% RSLogix 500 project HB_1_Filler.RSS, saved by version 12.00.00.00 %
PROJECT "PLC"    % processor: MicroLogix 1400 %

PROGRAM FILES
  LAD 2 "MAIN"  23 rungs
  LAD 9 "DPSTR REAR"  42 rungs
  LAD 11 "MAP DI"  37 rungs
  LAD 12 "MAP DO"  17 rungs
  LAD 14 "ALARMS"  17 rungs

DATA FILES
  O0 OUTPUT  7 elements
  I1 INPUT  9 elements
  S2 STATUS  66 elements
  B3 BINARY  14 elements
  T4 TIMER  22 elements
  C5 COUNTER  10 elements
  R6 CONTROL  5 elements
  N7 INTEGER  50 elements
  F8 FLOAT  40 elements
  B11 MAP DI  5 elements
  B12 MAP DO  10 elements
  B13 FORCE OUT  10 elements
  B23 TYPICAL  30 elements
  T24 TYPICAL  90 elements
  C25 TYPICAL  10 elements
  N27 TYPICAL  200 elements
  F28 TYPICAL  40 elements

LADDER 2 "MAIN"
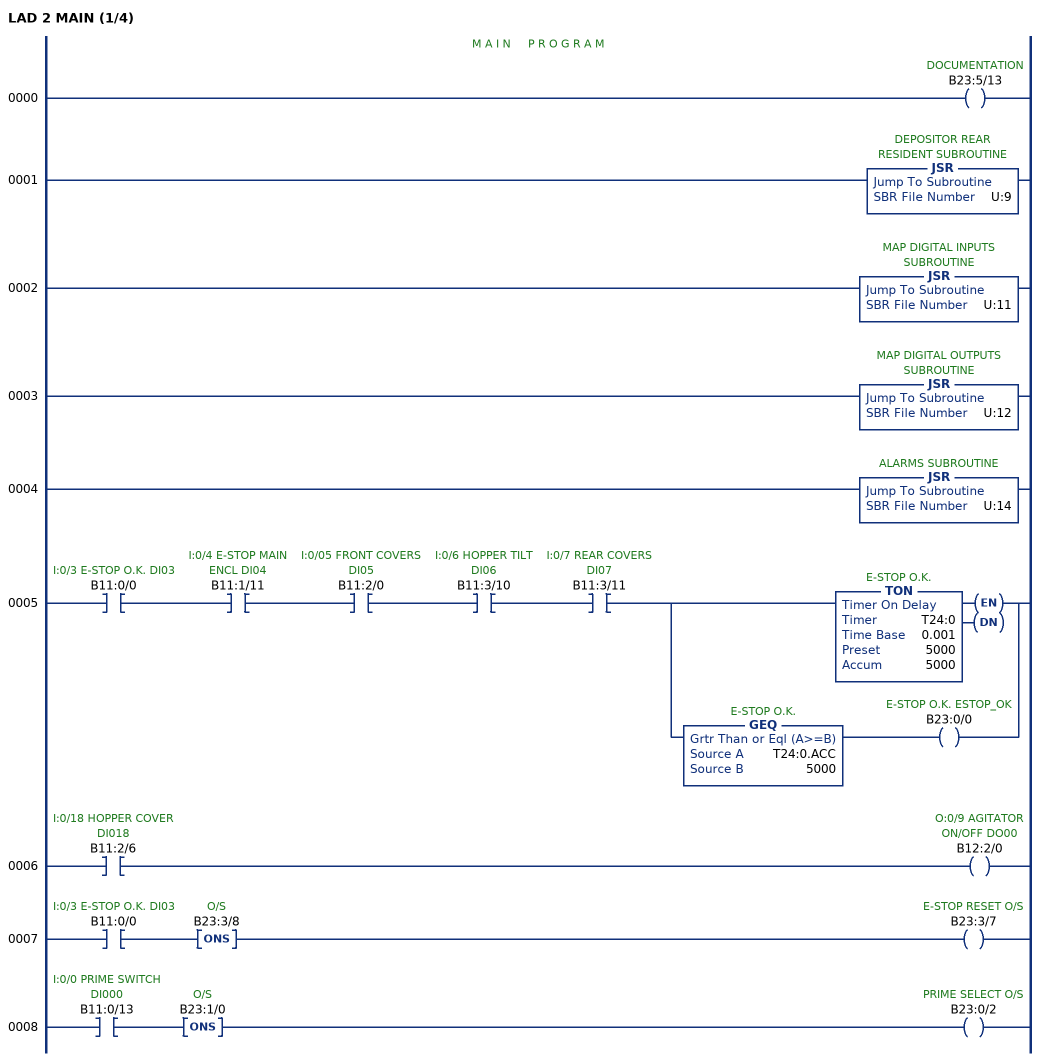
% Rung: 0 %
%  M A I N     P R O G R A M %
SOR OTE B23:5/13 EOR
%   B23:5/13  "DOCUMENTATION" %
% Rung: 1 %
SOR JSR U:9 EOR
%   U:9  "DEPOSITOR REAR RESIDENT SUBROUTINE" %
% Rung: 2 %
SOR JSR U:11 EOR
%   U:11  "MAP DIGITAL INPUTS SUBROUTINE" %
% Rung: 3 %
SOR JSR U:12 EOR
%   U:12  "MAP DIGITAL OUTPUTS SUBROUTINE" %
% Rung: 4 %
SOR JSR U:14 EOR
%   U:14  "ALARMS SUBROUTINE" %
% Rung: 5 %
SOR XIC B11:0/0 XIC B11:1/11 XIC B11:2/0 XIC B11:3/10 XIC B11:3/11 BST TON T24:0 0.001 5000 5000 NXB GEQ T24:0.ACC 5000 OTE B23:0/0 BND EOR
%   B11:0/0  DI03  "I:0/3 E-STOP O.K." %
%   B11:1/11  DI04  "I:0/4 E-STOP MAIN ENCL" %
%   B11:2/0  DI05  "I:0/05 FRONT COVERS" %
%   B11:3/10  DI06  "I:0/6 HOPPER TILT" %
%   B11:3/11  DI07  "I:0/7 REAR COVERS" %
%   T24:0  "E-STOP O.K." %
%   B23:0/0  ESTOP_OK  "E-STOP O.K." %
% Rung: 6 %
SOR XIC B11:2/6 OTE B12:2/0 EOR
%   B11:2/6  DI018  "I:0/18 HOPPER COVER" %
%   B12:2/0  DO00  "O:0/9 AGITATOR ON/OFF" %
% Rung: 7 %
SOR XIC B11:0/0 ONS B23:3/8 OTE B23:3/7 EOR
%   B11:0/0  DI03  "I:0/3 E-STOP O.K." %
%   B23:3/8  "O/S" %
%   B23:3/7  "E-STOP RESET O/S" %
% Rung: 8 %
SOR XIC B11:0/13 ONS B23:1/0 OTE B23:0/2 EOR
%   B11:0/13  DI000  "I:0/0 PRIME SWITCH" %
%   B23:1/0  "O/S" %
%   B23:0/2  "PRIME SELECT O/S" %

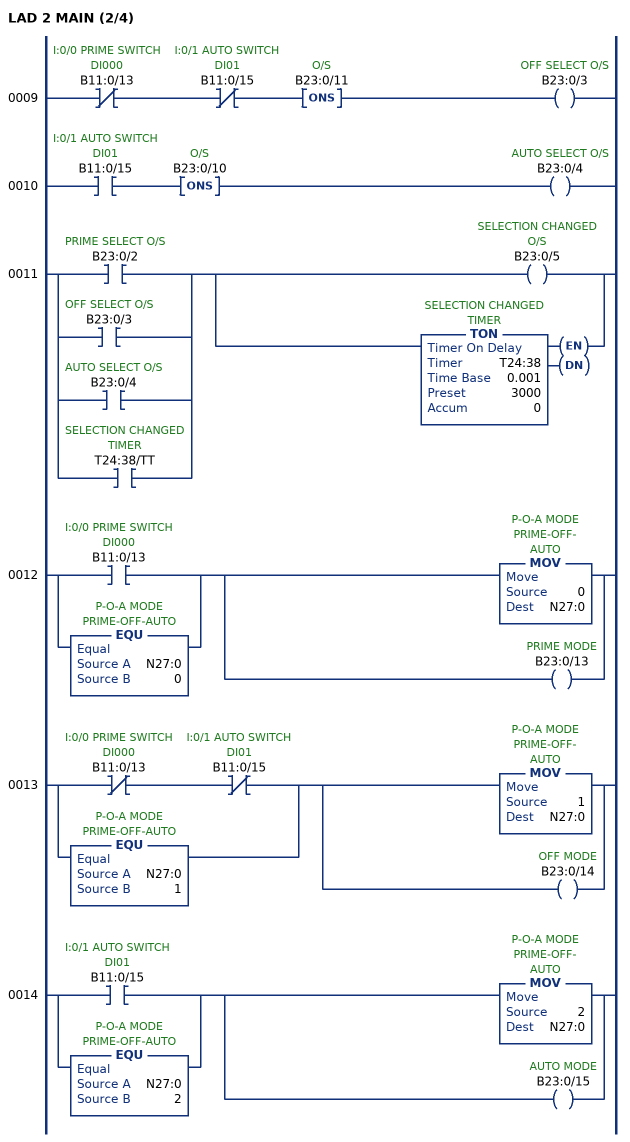
% Rung: 9 %
SOR XIO B11:0/13 XIO B11:0/15 ONS B23:0/11 OTE B23:0/3 EOR
%   B11:0/13  DI000  "I:0/0 PRIME SWITCH" %
%   B11:0/15  DI01  "I:0/1 AUTO SWITCH" %
%   B23:0/11  "O/S" %
%   B23:0/3  "OFF SELECT O/S" %
% Rung: 10 %
SOR XIC B11:0/15 ONS B23:0/10 OTE B23:0/4 EOR
%   B11:0/15  DI01  "I:0/1 AUTO SWITCH" %
%   B23:0/10  "O/S" %
%   B23:0/4  "AUTO SELECT O/S" %
% Rung: 11 %
SOR BST XIC B23:0/2 NXB XIC B23:0/3 NXB XIC B23:0/4 NXB XIC T24:38/TT BND BST OTE B23:0/5 NXB TON T24:38 0.001 3000 0 BND EOR
%   B23:0/2  "PRIME SELECT O/S" %
%   B23:0/3  "OFF SELECT O/S" %
%   B23:0/4  "AUTO SELECT O/S" %
%   T24:38  "SELECTION CHANGED TIMER" %
%   B23:0/5  "SELECTION CHANGED O/S" %
% Rung: 12 %
SOR BST XIC B11:0/13 NXB EQU N27:0 0 BND BST MOV 0 N27:0 NXB OTE B23:0/13 BND EOR
%   B11:0/13  DI000  "I:0/0 PRIME SWITCH" %
%   N27:0  "P-O-A MODE PRIME-OFF-AUTO" %
%   B23:0/13  "PRIME MODE" %
% Rung: 13 %
SOR BST XIO B11:0/13 XIO B11:0/15 NXB EQU N27:0 1 BND BST MOV 1 N27:0 NXB OTE B23:0/14 BND EOR
%   B11:0/13  DI000  "I:0/0 PRIME SWITCH" %
%   B11:0/15  DI01  "I:0/1 AUTO SWITCH" %
%   N27:0  "P-O-A MODE PRIME-OFF-AUTO" %
%   B23:0/14  "OFF MODE" %
% Rung: 14 %
SOR BST XIC B11:0/15 NXB EQU N27:0 2 BND BST MOV 2 N27:0 NXB OTE B23:0/15 BND EOR
%   B11:0/15  DI01  "I:0/1 AUTO SWITCH" %
%   N27:0  "P-O-A MODE PRIME-OFF-AUTO" %
%   B23:0/15  "AUTO MODE" %

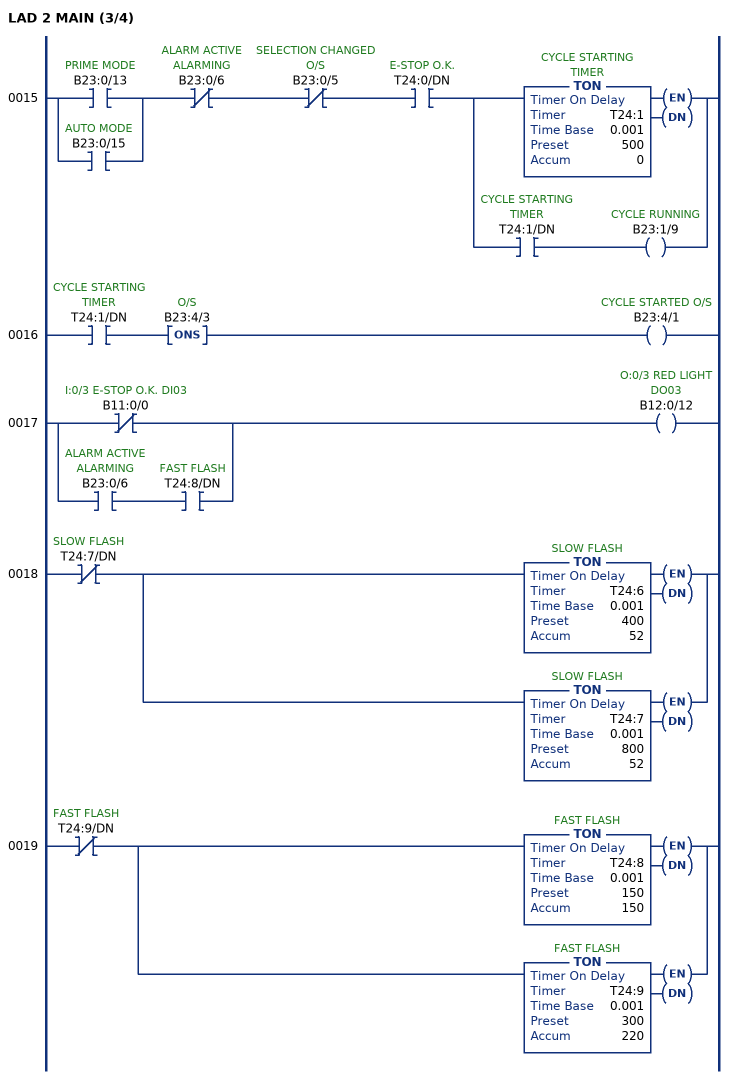
% Rung: 15 %
SOR BST XIC B23:0/13 NXB XIC B23:0/15 BND XIO B23:0/6 XIO B23:0/5 XIC T24:0/DN BST TON T24:1 0.001 500 0 NXB XIC T24:1/DN OTE B23:1/9 BND EOR
%   B23:0/13  "PRIME MODE" %
%   B23:0/15  "AUTO MODE" %
%   B23:0/6  ALARMING  "ALARM ACTIVE" %
%   B23:0/5  "SELECTION CHANGED O/S" %
%   T24:0  "E-STOP O.K." %
%   T24:1  "CYCLE STARTING TIMER" %
%   B23:1/9  "CYCLE RUNNING" %
% Rung: 16 %
SOR XIC T24:1/DN ONS B23:4/3 OTE B23:4/1 EOR
%   T24:1  "CYCLE STARTING TIMER" %
%   B23:4/3  "O/S" %
%   B23:4/1  "CYCLE STARTED O/S" %
% Rung: 17 %
SOR BST XIO B11:0/0 NXB XIC B23:0/6 XIC T24:8/DN BND OTE B12:0/12 EOR
%   B11:0/0  DI03  "I:0/3 E-STOP O.K." %
%   B23:0/6  ALARMING  "ALARM ACTIVE" %
%   T24:8  "FAST FLASH" %
%   B12:0/12  DO03  "O:0/3 RED LIGHT" %
% Rung: 18 %
SOR XIO T24:7/DN BST TON T24:6 0.001 400 52 NXB TON T24:7 0.001 800 52 BND EOR
%   T24:7  "SLOW FLASH" %
%   T24:6  "SLOW FLASH" %
% Rung: 19 %
SOR XIO T24:9/DN BST TON T24:8 0.001 150 150 NXB TON T24:9 0.001 300 220 BND EOR
%   T24:9  "FAST FLASH" %
%   T24:8  "FAST FLASH" %

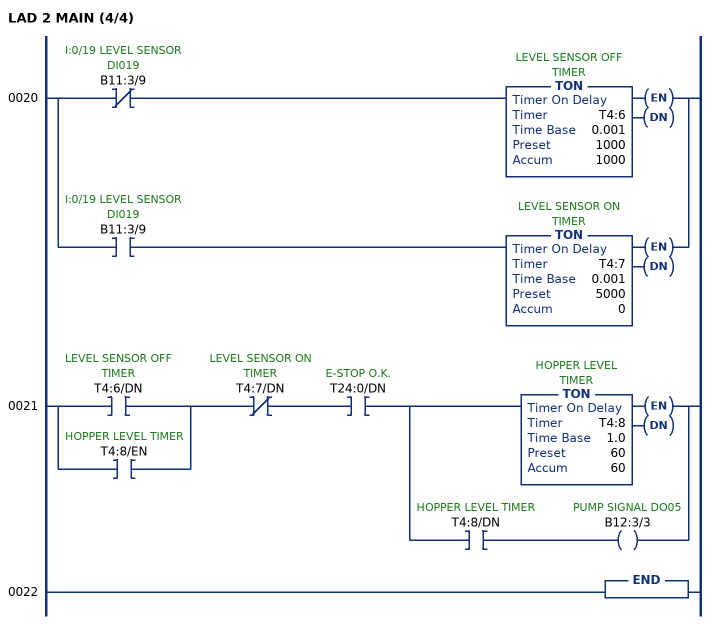
% Rung: 20 %
SOR BST XIO B11:3/9 TON T4:6 0.001 1000 1000 NXB XIC B11:3/9 TON T4:7 0.001 5000 0 BND EOR
%   B11:3/9  DI019  "I:0/19 LEVEL SENSOR" %
%   T4:6  "LEVEL SENSOR OFF TIMER" %
%   T4:7  "LEVEL SENSOR ON TIMER" %
% Rung: 21 %
SOR BST XIC T4:6/DN NXB XIC T4:8/EN BND XIO T4:7/DN XIC T24:0/DN BST TON T4:8 1.0 60 60 NXB XIC T4:8/DN OTE B12:3/3 BND EOR
%   T4:6  "LEVEL SENSOR OFF TIMER" %
%   T4:8  "HOPPER LEVEL TIMER" %
%   T4:7  "LEVEL SENSOR ON TIMER" %
%   T24:0  "E-STOP O.K." %
%   B12:3/3  DO05  "PUMP SIGNAL" %
% Rung: 22 %
SOR END EOR

LADDER 9 "DPSTR REAR"
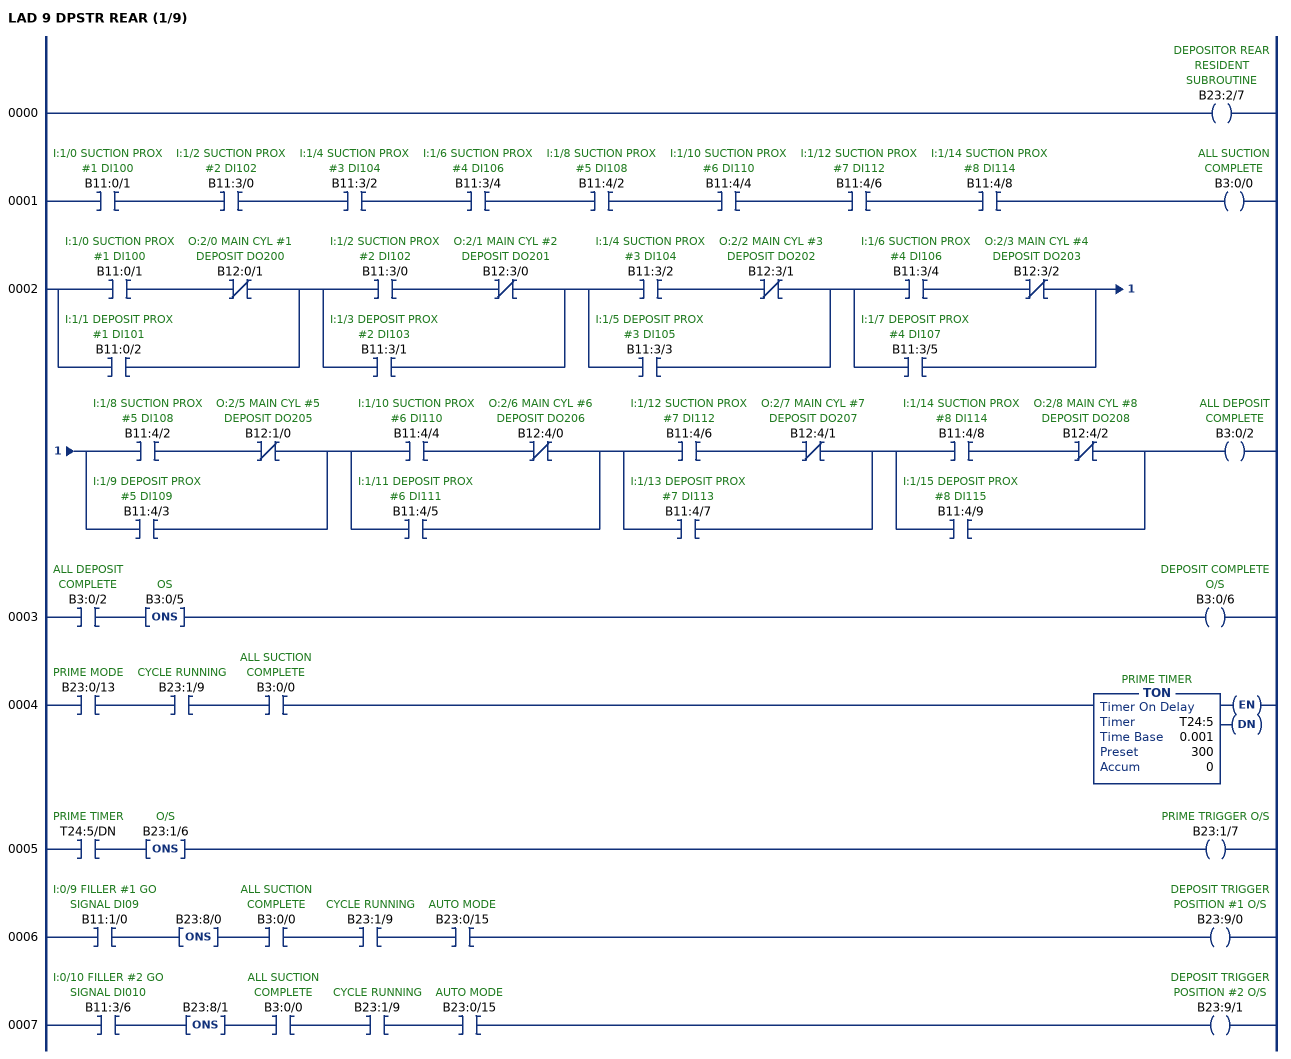
% Rung: 0 %
SOR OTE B23:2/7 EOR
%   B23:2/7  "DEPOSITOR REAR RESIDENT SUBROUTINE" %
% Rung: 1 %
SOR XIC B11:0/1 XIC B11:3/0 XIC B11:3/2 XIC B11:3/4 XIC B11:4/2 XIC B11:4/4 XIC B11:4/6 XIC B11:4/8 OTE B3:0/0 EOR
%   B11:0/1  DI100  "I:1/0 SUCTION PROX #1" %
%   B11:3/0  DI102  "I:1/2 SUCTION PROX #2" %
%   B11:3/2  DI104  "I:1/4 SUCTION PROX #3" %
%   B11:3/4  DI106  "I:1/6 SUCTION PROX #4" %
%   B11:4/2  DI108  "I:1/8 SUCTION PROX #5" %
%   B11:4/4  DI110  "I:1/10 SUCTION PROX #6" %
%   B11:4/6  DI112  "I:1/12 SUCTION PROX #7" %
%   B11:4/8  DI114  "I:1/14 SUCTION PROX #8" %
%   B3:0/0  "ALL SUCTION COMPLETE" %
% Rung: 2 %
SOR BST XIC B11:0/1 XIO B12:0/1 NXB XIC B11:0/2 BND BST XIC B11:3/0 XIO B12:3/0 NXB XIC B11:3/1 BND BST XIC B11:3/2 XIO B12:3/1 NXB XIC B11:3/3 BND BST XIC B11:3/4 XIO B12:3/2 NXB XIC B11:3/5 BND BST XIC B11:4/2 XIO B12:1/0 NXB XIC B11:4/3 BND BST XIC B11:4/4 XIO B12:4/0 NXB XIC B11:4/5 BND BST XIC B11:4/6 XIO B12:4/1 NXB XIC B11:4/7 BND BST XIC B11:4/8 XIO B12:4/2 NXB XIC B11:4/9 BND OTE B3:0/2 EOR
%   B11:0/1  DI100  "I:1/0 SUCTION PROX #1" %
%   B12:0/1  DO200  "O:2/0 MAIN CYL #1 DEPOSIT" %
%   B11:0/2  DI101  "I:1/1 DEPOSIT PROX #1" %
%   B11:3/0  DI102  "I:1/2 SUCTION PROX #2" %
%   B12:3/0  DO201  "O:2/1 MAIN CYL #2 DEPOSIT" %
%   B11:3/1  DI103  "I:1/3 DEPOSIT PROX #2" %
%   B11:3/2  DI104  "I:1/4 SUCTION PROX #3" %
%   B12:3/1  DO202  "O:2/2 MAIN CYL #3 DEPOSIT" %
%   B11:3/3  DI105  "I:1/5 DEPOSIT PROX #3" %
%   B11:3/4  DI106  "I:1/6 SUCTION PROX #4" %
%   B12:3/2  DO203  "O:2/3 MAIN CYL #4 DEPOSIT" %
%   B11:3/5  DI107  "I:1/7 DEPOSIT PROX #4" %
%   B11:4/2  DI108  "I:1/8 SUCTION PROX #5" %
%   B12:1/0  DO205  "O:2/5 MAIN CYL #5 DEPOSIT" %
%   B11:4/3  DI109  "I:1/9 DEPOSIT PROX #5" %
%   B11:4/4  DI110  "I:1/10 SUCTION PROX #6" %
%   B12:4/0  DO206  "O:2/6 MAIN CYL #6 DEPOSIT" %
%   B11:4/5  DI111  "I:1/11 DEPOSIT PROX #6" %
%   B11:4/6  DI112  "I:1/12 SUCTION PROX #7" %
%   B12:4/1  DO207  "O:2/7 MAIN CYL #7 DEPOSIT" %
%   B11:4/7  DI113  "I:1/13 DEPOSIT PROX #7" %
%   B11:4/8  DI114  "I:1/14 SUCTION PROX #8" %
%   B12:4/2  DO208  "O:2/8 MAIN CYL #8 DEPOSIT" %
%   B11:4/9  DI115  "I:1/15 DEPOSIT PROX #8" %
%   B3:0/2  "ALL DEPOSIT COMPLETE" %
% Rung: 3 %
SOR XIC B3:0/2 ONS B3:0/5 OTE B3:0/6 EOR
%   B3:0/2  "ALL DEPOSIT COMPLETE" %
%   B3:0/5  "OS" %
%   B3:0/6  "DEPOSIT COMPLETE O/S" %
% Rung: 4 %
SOR XIC B23:0/13 XIC B23:1/9 XIC B3:0/0 TON T24:5 0.001 300 0 EOR
%   B23:0/13  "PRIME MODE" %
%   B23:1/9  "CYCLE RUNNING" %
%   B3:0/0  "ALL SUCTION COMPLETE" %
%   T24:5  "PRIME TIMER" %
% Rung: 5 %
SOR XIC T24:5/DN ONS B23:1/6 OTE B23:1/7 EOR
%   T24:5  "PRIME TIMER" %
%   B23:1/6  "O/S" %
%   B23:1/7  "PRIME TRIGGER O/S" %
% Rung: 6 %
SOR XIC B11:1/0 ONS B23:8/0 XIC B3:0/0 XIC B23:1/9 XIC B23:0/15 OTE B23:9/0 EOR
%   B11:1/0  DI09  "I:0/9 FILLER #1 GO SIGNAL" %
%   B3:0/0  "ALL SUCTION COMPLETE" %
%   B23:1/9  "CYCLE RUNNING" %
%   B23:0/15  "AUTO MODE" %
%   B23:9/0  "DEPOSIT TRIGGER POSITION #1 O/S" %
% Rung: 7 %
SOR XIC B11:3/6 ONS B23:8/1 XIC B3:0/0 XIC B23:1/9 XIC B23:0/15 OTE B23:9/1 EOR
%   B11:3/6  DI010  "I:0/10 FILLER #2 GO SIGNAL" %
%   B3:0/0  "ALL SUCTION COMPLETE" %
%   B23:1/9  "CYCLE RUNNING" %
%   B23:0/15  "AUTO MODE" %
%   B23:9/1  "DEPOSIT TRIGGER POSITION #2 O/S" %

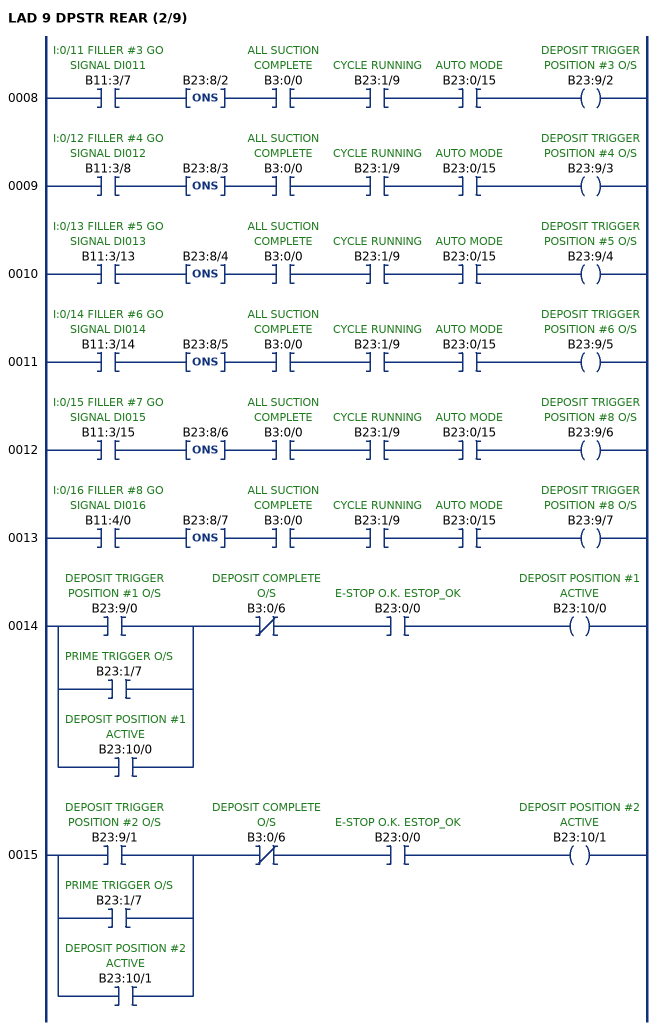
% Rung: 8 %
SOR XIC B11:3/7 ONS B23:8/2 XIC B3:0/0 XIC B23:1/9 XIC B23:0/15 OTE B23:9/2 EOR
%   B11:3/7  DI011  "I:0/11 FILLER #3 GO SIGNAL" %
%   B3:0/0  "ALL SUCTION COMPLETE" %
%   B23:1/9  "CYCLE RUNNING" %
%   B23:0/15  "AUTO MODE" %
%   B23:9/2  "DEPOSIT TRIGGER POSITION #3 O/S" %
% Rung: 9 %
SOR XIC B11:3/8 ONS B23:8/3 XIC B3:0/0 XIC B23:1/9 XIC B23:0/15 OTE B23:9/3 EOR
%   B11:3/8  DI012  "I:0/12 FILLER #4 GO SIGNAL" %
%   B3:0/0  "ALL SUCTION COMPLETE" %
%   B23:1/9  "CYCLE RUNNING" %
%   B23:0/15  "AUTO MODE" %
%   B23:9/3  "DEPOSIT TRIGGER POSITION #4 O/S" %
% Rung: 10 %
SOR XIC B11:3/13 ONS B23:8/4 XIC B3:0/0 XIC B23:1/9 XIC B23:0/15 OTE B23:9/4 EOR
%   B11:3/13  DI013  "I:0/13 FILLER #5 GO SIGNAL" %
%   B3:0/0  "ALL SUCTION COMPLETE" %
%   B23:1/9  "CYCLE RUNNING" %
%   B23:0/15  "AUTO MODE" %
%   B23:9/4  "DEPOSIT TRIGGER POSITION #5 O/S" %
% Rung: 11 %
SOR XIC B11:3/14 ONS B23:8/5 XIC B3:0/0 XIC B23:1/9 XIC B23:0/15 OTE B23:9/5 EOR
%   B11:3/14  DI014  "I:0/14 FILLER #6 GO SIGNAL" %
%   B3:0/0  "ALL SUCTION COMPLETE" %
%   B23:1/9  "CYCLE RUNNING" %
%   B23:0/15  "AUTO MODE" %
%   B23:9/5  "DEPOSIT TRIGGER POSITION #6 O/S" %
% Rung: 12 %
SOR XIC B11:3/15 ONS B23:8/6 XIC B3:0/0 XIC B23:1/9 XIC B23:0/15 OTE B23:9/6 EOR
%   B11:3/15  DI015  "I:0/15 FILLER #7 GO SIGNAL" %
%   B3:0/0  "ALL SUCTION COMPLETE" %
%   B23:1/9  "CYCLE RUNNING" %
%   B23:0/15  "AUTO MODE" %
%   B23:9/6  "DEPOSIT TRIGGER POSITION #8 O/S" %
% Rung: 13 %
SOR XIC B11:4/0 ONS B23:8/7 XIC B3:0/0 XIC B23:1/9 XIC B23:0/15 OTE B23:9/7 EOR
%   B11:4/0  DI016  "I:0/16 FILLER #8 GO SIGNAL" %
%   B3:0/0  "ALL SUCTION COMPLETE" %
%   B23:1/9  "CYCLE RUNNING" %
%   B23:0/15  "AUTO MODE" %
%   B23:9/7  "DEPOSIT TRIGGER POSITION #8 O/S" %
% Rung: 14 %
SOR BST XIC B23:9/0 NXB XIC B23:1/7 NXB XIC B23:10/0 BND XIO B3:0/6 XIC B23:0/0 OTE B23:10/0 EOR
%   B23:9/0  "DEPOSIT TRIGGER POSITION #1 O/S" %
%   B23:1/7  "PRIME TRIGGER O/S" %
%   B23:10/0  "DEPOSIT POSITION #1 ACTIVE" %
%   B3:0/6  "DEPOSIT COMPLETE O/S" %
%   B23:0/0  ESTOP_OK  "E-STOP O.K." %
% Rung: 15 %
SOR BST XIC B23:9/1 NXB XIC B23:1/7 NXB XIC B23:10/1 BND XIO B3:0/6 XIC B23:0/0 OTE B23:10/1 EOR
%   B23:9/1  "DEPOSIT TRIGGER POSITION #2 O/S" %
%   B23:1/7  "PRIME TRIGGER O/S" %
%   B23:10/1  "DEPOSIT POSITION #2 ACTIVE" %
%   B3:0/6  "DEPOSIT COMPLETE O/S" %
%   B23:0/0  ESTOP_OK  "E-STOP O.K." %

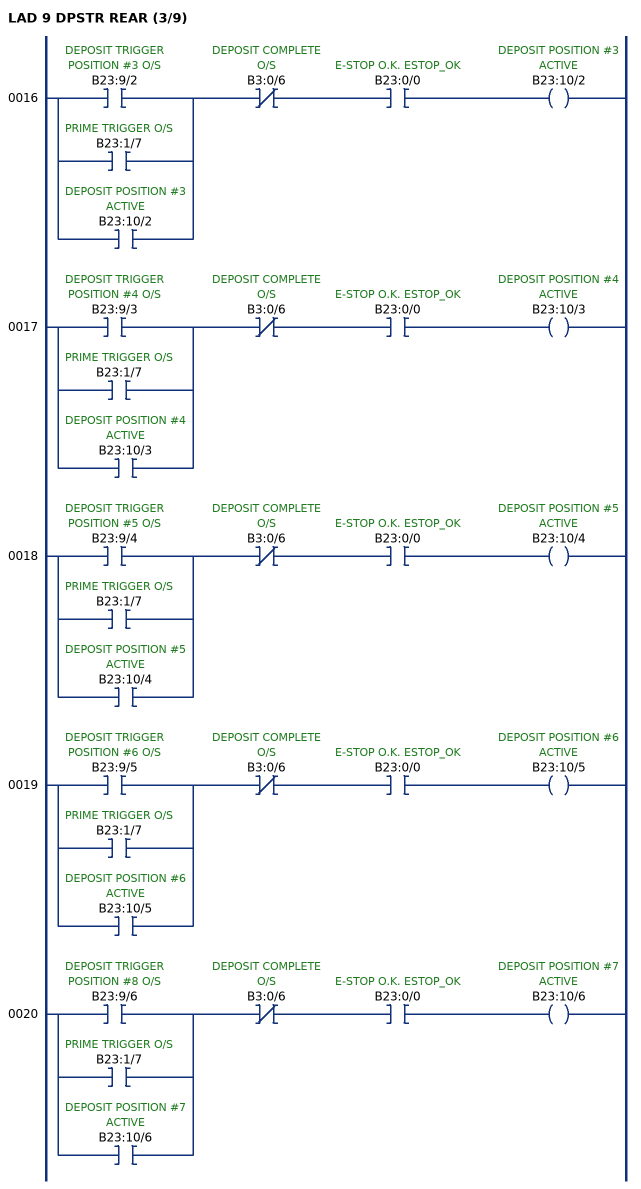
% Rung: 16 %
SOR BST XIC B23:9/2 NXB XIC B23:1/7 NXB XIC B23:10/2 BND XIO B3:0/6 XIC B23:0/0 OTE B23:10/2 EOR
%   B23:9/2  "DEPOSIT TRIGGER POSITION #3 O/S" %
%   B23:1/7  "PRIME TRIGGER O/S" %
%   B23:10/2  "DEPOSIT POSITION #3 ACTIVE" %
%   B3:0/6  "DEPOSIT COMPLETE O/S" %
%   B23:0/0  ESTOP_OK  "E-STOP O.K." %
% Rung: 17 %
SOR BST XIC B23:9/3 NXB XIC B23:1/7 NXB XIC B23:10/3 BND XIO B3:0/6 XIC B23:0/0 OTE B23:10/3 EOR
%   B23:9/3  "DEPOSIT TRIGGER POSITION #4 O/S" %
%   B23:1/7  "PRIME TRIGGER O/S" %
%   B23:10/3  "DEPOSIT POSITION #4 ACTIVE" %
%   B3:0/6  "DEPOSIT COMPLETE O/S" %
%   B23:0/0  ESTOP_OK  "E-STOP O.K." %
% Rung: 18 %
SOR BST XIC B23:9/4 NXB XIC B23:1/7 NXB XIC B23:10/4 BND XIO B3:0/6 XIC B23:0/0 OTE B23:10/4 EOR
%   B23:9/4  "DEPOSIT TRIGGER POSITION #5 O/S" %
%   B23:1/7  "PRIME TRIGGER O/S" %
%   B23:10/4  "DEPOSIT POSITION #5 ACTIVE" %
%   B3:0/6  "DEPOSIT COMPLETE O/S" %
%   B23:0/0  ESTOP_OK  "E-STOP O.K." %
% Rung: 19 %
SOR BST XIC B23:9/5 NXB XIC B23:1/7 NXB XIC B23:10/5 BND XIO B3:0/6 XIC B23:0/0 OTE B23:10/5 EOR
%   B23:9/5  "DEPOSIT TRIGGER POSITION #6 O/S" %
%   B23:1/7  "PRIME TRIGGER O/S" %
%   B23:10/5  "DEPOSIT POSITION #6 ACTIVE" %
%   B3:0/6  "DEPOSIT COMPLETE O/S" %
%   B23:0/0  ESTOP_OK  "E-STOP O.K." %
% Rung: 20 %
SOR BST XIC B23:9/6 NXB XIC B23:1/7 NXB XIC B23:10/6 BND XIO B3:0/6 XIC B23:0/0 OTE B23:10/6 EOR
%   B23:9/6  "DEPOSIT TRIGGER POSITION #8 O/S" %
%   B23:1/7  "PRIME TRIGGER O/S" %
%   B23:10/6  "DEPOSIT POSITION #7 ACTIVE" %
%   B3:0/6  "DEPOSIT COMPLETE O/S" %
%   B23:0/0  ESTOP_OK  "E-STOP O.K." %

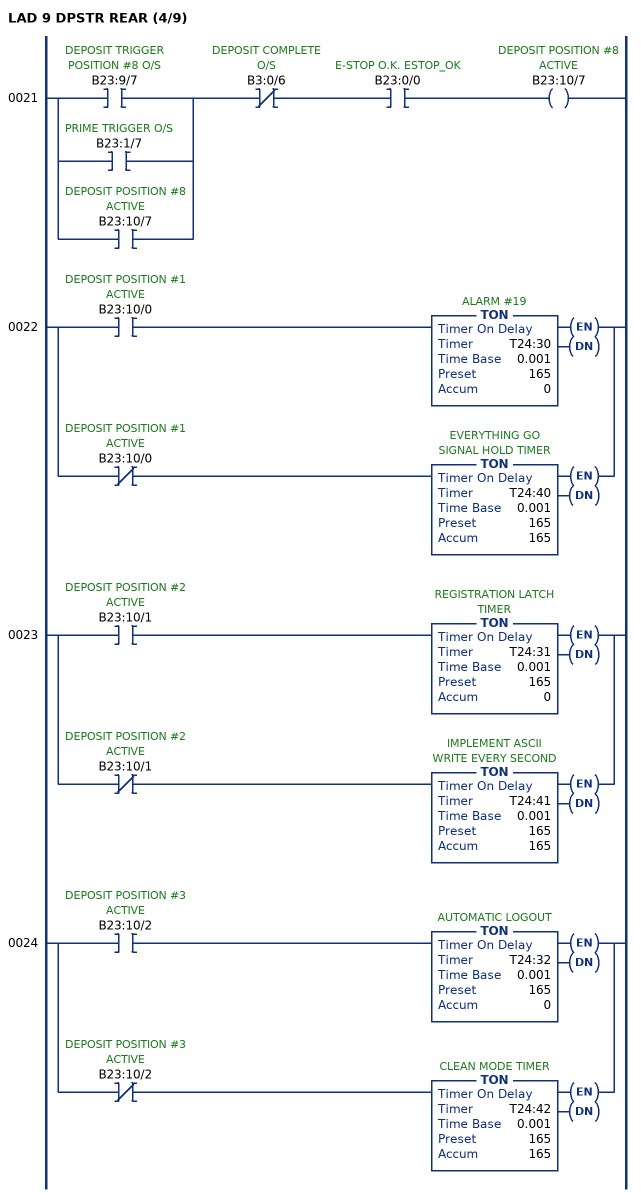
% Rung: 21 %
SOR BST XIC B23:9/7 NXB XIC B23:1/7 NXB XIC B23:10/7 BND XIO B3:0/6 XIC B23:0/0 OTE B23:10/7 EOR
%   B23:9/7  "DEPOSIT TRIGGER POSITION #8 O/S" %
%   B23:1/7  "PRIME TRIGGER O/S" %
%   B23:10/7  "DEPOSIT POSITION #8 ACTIVE" %
%   B3:0/6  "DEPOSIT COMPLETE O/S" %
%   B23:0/0  ESTOP_OK  "E-STOP O.K." %
% Rung: 22 %
SOR BST XIC B23:10/0 TON T24:30 0.001 165 0 NXB XIO B23:10/0 TON T24:40 0.001 165 165 BND EOR
%   B23:10/0  "DEPOSIT POSITION #1 ACTIVE" %
%   T24:30  "ALARM #19" %
%   T24:40  "EVERYTHING GO SIGNAL HOLD TIMER" %
% Rung: 23 %
SOR BST XIC B23:10/1 TON T24:31 0.001 165 0 NXB XIO B23:10/1 TON T24:41 0.001 165 165 BND EOR
%   B23:10/1  "DEPOSIT POSITION #2 ACTIVE" %
%   T24:31  "REGISTRATION LATCH TIMER" %
%   T24:41  "IMPLEMENT ASCII WRITE EVERY SECOND" %
% Rung: 24 %
SOR BST XIC B23:10/2 TON T24:32 0.001 165 0 NXB XIO B23:10/2 TON T24:42 0.001 165 165 BND EOR
%   B23:10/2  "DEPOSIT POSITION #3 ACTIVE" %
%   T24:32  "AUTOMATIC LOGOUT" %
%   T24:42  "CLEAN MODE TIMER" %

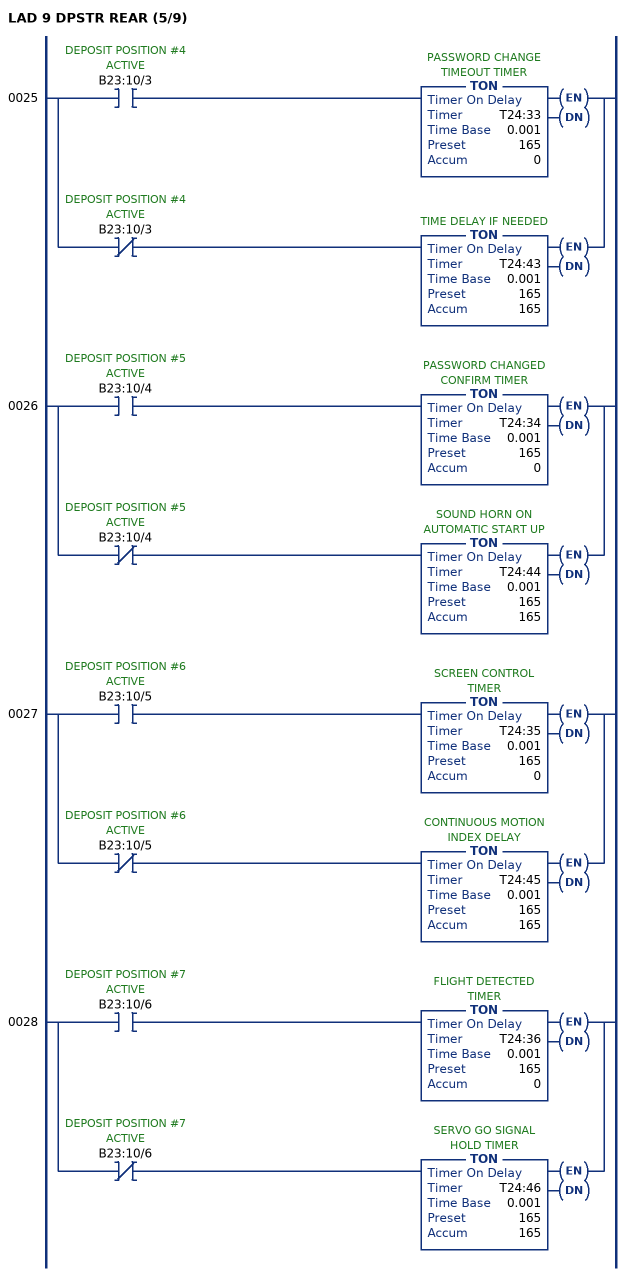
% Rung: 25 %
SOR BST XIC B23:10/3 TON T24:33 0.001 165 0 NXB XIO B23:10/3 TON T24:43 0.001 165 165 BND EOR
%   B23:10/3  "DEPOSIT POSITION #4 ACTIVE" %
%   T24:33  "PASSWORD CHANGE TIMEOUT TIMER" %
%   T24:43  "TIME DELAY IF NEEDED" %
% Rung: 26 %
SOR BST XIC B23:10/4 TON T24:34 0.001 165 0 NXB XIO B23:10/4 TON T24:44 0.001 165 165 BND EOR
%   B23:10/4  "DEPOSIT POSITION #5 ACTIVE" %
%   T24:34  "PASSWORD CHANGED CONFIRM TIMER" %
%   T24:44  "SOUND HORN ON AUTOMATIC START UP" %
% Rung: 27 %
SOR BST XIC B23:10/5 TON T24:35 0.001 165 0 NXB XIO B23:10/5 TON T24:45 0.001 165 165 BND EOR
%   B23:10/5  "DEPOSIT POSITION #6 ACTIVE" %
%   T24:35  "SCREEN CONTROL TIMER" %
%   T24:45  "CONTINUOUS MOTION INDEX DELAY" %
% Rung: 28 %
SOR BST XIC B23:10/6 TON T24:36 0.001 165 0 NXB XIO B23:10/6 TON T24:46 0.001 165 165 BND EOR
%   B23:10/6  "DEPOSIT POSITION #7 ACTIVE" %
%   T24:36  "FLIGHT DETECTED TIMER" %
%   T24:46  "SERVO GO SIGNAL HOLD TIMER" %

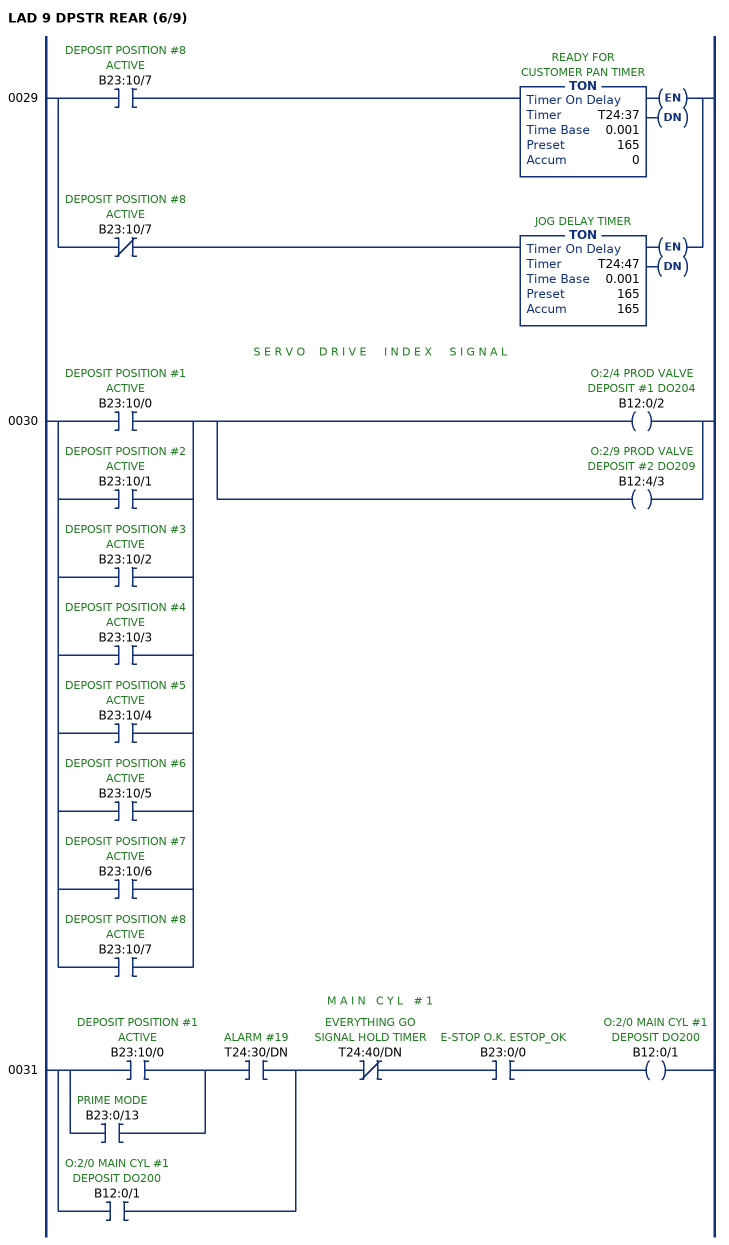
% Rung: 29 %
SOR BST XIC B23:10/7 TON T24:37 0.001 165 0 NXB XIO B23:10/7 TON T24:47 0.001 165 165 BND EOR
%   B23:10/7  "DEPOSIT POSITION #8 ACTIVE" %
%   T24:37  "READY FOR CUSTOMER PAN TIMER" %
%   T24:47  "JOG DELAY TIMER" %
% Rung: 30 %
%     S E R V O    D R I V E     I N D E X     S I G N A L %
SOR BST XIC B23:10/0 NXB XIC B23:10/1 NXB XIC B23:10/2 NXB XIC B23:10/3 NXB XIC B23:10/4 NXB XIC B23:10/5 NXB XIC B23:10/6 NXB XIC B23:10/7 BND BST OTE B12:0/2 NXB OTE B12:4/3 BND EOR
%   B23:10/0  "DEPOSIT POSITION #1 ACTIVE" %
%   B23:10/1  "DEPOSIT POSITION #2 ACTIVE" %
%   B23:10/2  "DEPOSIT POSITION #3 ACTIVE" %
%   B23:10/3  "DEPOSIT POSITION #4 ACTIVE" %
%   B23:10/4  "DEPOSIT POSITION #5 ACTIVE" %
%   B23:10/5  "DEPOSIT POSITION #6 ACTIVE" %
%   B23:10/6  "DEPOSIT POSITION #7 ACTIVE" %
%   B23:10/7  "DEPOSIT POSITION #8 ACTIVE" %
%   B12:0/2  DO204  "O:2/4 PROD VALVE DEPOSIT #1" %
%   B12:4/3  DO209  "O:2/9 PROD VALVE DEPOSIT #2" %
% Rung: 31 %
%     M A I N   C Y L   # 1 %
SOR BST BST XIC B23:10/0 NXB XIC B23:0/13 BND XIC T24:30/DN NXB XIC B12:0/1 BND XIO T24:40/DN XIC B23:0/0 OTE B12:0/1 EOR
%   B23:10/0  "DEPOSIT POSITION #1 ACTIVE" %
%   B23:0/13  "PRIME MODE" %
%   T24:30  "ALARM #19" %
%   B12:0/1  DO200  "O:2/0 MAIN CYL #1 DEPOSIT" %
%   T24:40  "EVERYTHING GO SIGNAL HOLD TIMER" %
%   B23:0/0  ESTOP_OK  "E-STOP O.K." %

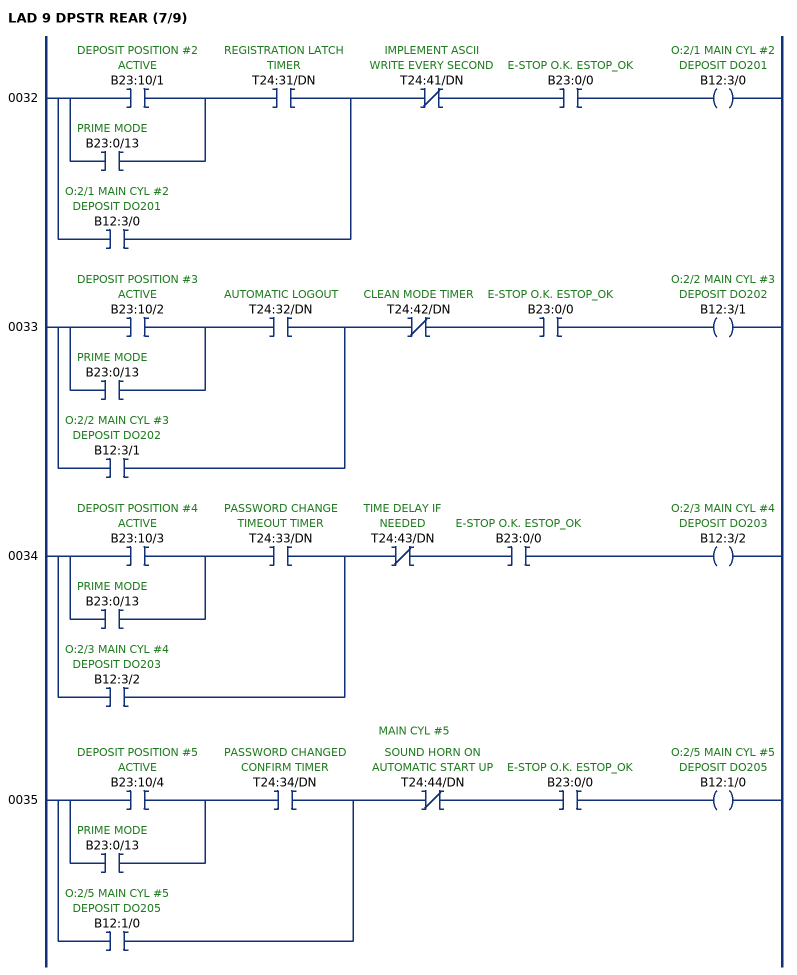
% Rung: 32 %
SOR BST BST XIC B23:10/1 NXB XIC B23:0/13 BND XIC T24:31/DN NXB XIC B12:3/0 BND XIO T24:41/DN XIC B23:0/0 OTE B12:3/0 EOR
%   B23:10/1  "DEPOSIT POSITION #2 ACTIVE" %
%   B23:0/13  "PRIME MODE" %
%   T24:31  "REGISTRATION LATCH TIMER" %
%   B12:3/0  DO201  "O:2/1 MAIN CYL #2 DEPOSIT" %
%   T24:41  "IMPLEMENT ASCII WRITE EVERY SECOND" %
%   B23:0/0  ESTOP_OK  "E-STOP O.K." %
% Rung: 33 %
SOR BST BST XIC B23:10/2 NXB XIC B23:0/13 BND XIC T24:32/DN NXB XIC B12:3/1 BND XIO T24:42/DN XIC B23:0/0 OTE B12:3/1 EOR
%   B23:10/2  "DEPOSIT POSITION #3 ACTIVE" %
%   B23:0/13  "PRIME MODE" %
%   T24:32  "AUTOMATIC LOGOUT" %
%   B12:3/1  DO202  "O:2/2 MAIN CYL #3 DEPOSIT" %
%   T24:42  "CLEAN MODE TIMER" %
%   B23:0/0  ESTOP_OK  "E-STOP O.K." %
% Rung: 34 %
SOR BST BST XIC B23:10/3 NXB XIC B23:0/13 BND XIC T24:33/DN NXB XIC B12:3/2 BND XIO T24:43/DN XIC B23:0/0 OTE B12:3/2 EOR
%   B23:10/3  "DEPOSIT POSITION #4 ACTIVE" %
%   B23:0/13  "PRIME MODE" %
%   T24:33  "PASSWORD CHANGE TIMEOUT TIMER" %
%   B12:3/2  DO203  "O:2/3 MAIN CYL #4 DEPOSIT" %
%   T24:43  "TIME DELAY IF NEEDED" %
%   B23:0/0  ESTOP_OK  "E-STOP O.K." %
% Rung: 35 %
% MAIN CYL #5 %
SOR BST BST XIC B23:10/4 NXB XIC B23:0/13 BND XIC T24:34/DN NXB XIC B12:1/0 BND XIO T24:44/DN XIC B23:0/0 OTE B12:1/0 EOR
%   B23:10/4  "DEPOSIT POSITION #5 ACTIVE" %
%   B23:0/13  "PRIME MODE" %
%   T24:34  "PASSWORD CHANGED CONFIRM TIMER" %
%   B12:1/0  DO205  "O:2/5 MAIN CYL #5 DEPOSIT" %
%   T24:44  "SOUND HORN ON AUTOMATIC START UP" %
%   B23:0/0  ESTOP_OK  "E-STOP O.K." %

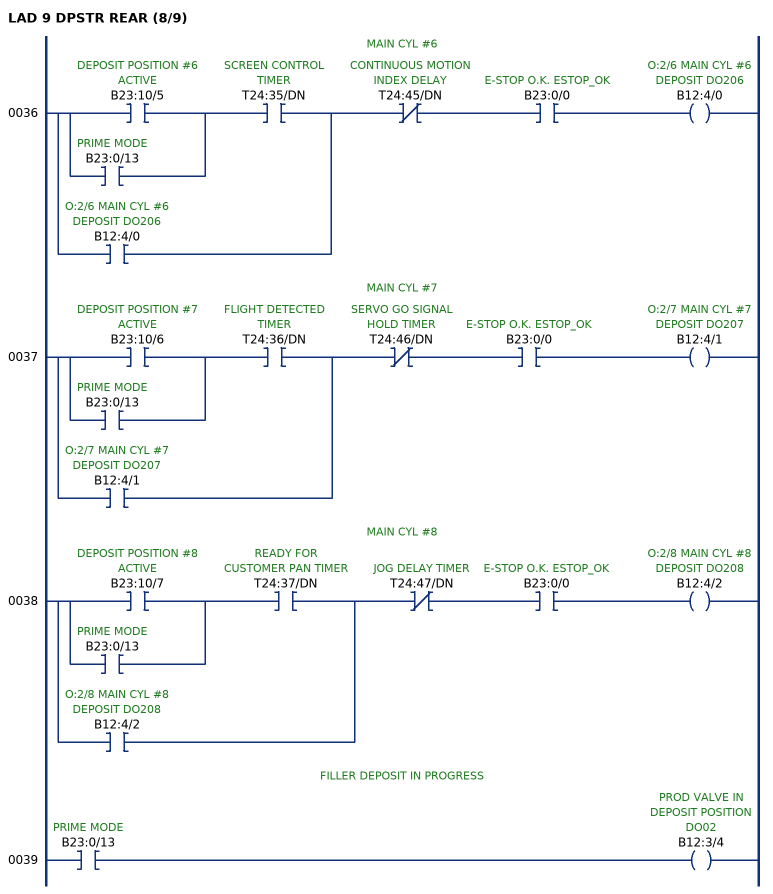
% Rung: 36 %
% MAIN CYL #6 %
SOR BST BST XIC B23:10/5 NXB XIC B23:0/13 BND XIC T24:35/DN NXB XIC B12:4/0 BND XIO T24:45/DN XIC B23:0/0 OTE B12:4/0 EOR
%   B23:10/5  "DEPOSIT POSITION #6 ACTIVE" %
%   B23:0/13  "PRIME MODE" %
%   T24:35  "SCREEN CONTROL TIMER" %
%   B12:4/0  DO206  "O:2/6 MAIN CYL #6 DEPOSIT" %
%   T24:45  "CONTINUOUS MOTION INDEX DELAY" %
%   B23:0/0  ESTOP_OK  "E-STOP O.K." %
% Rung: 37 %
% MAIN CYL #7 %
SOR BST BST XIC B23:10/6 NXB XIC B23:0/13 BND XIC T24:36/DN NXB XIC B12:4/1 BND XIO T24:46/DN XIC B23:0/0 OTE B12:4/1 EOR
%   B23:10/6  "DEPOSIT POSITION #7 ACTIVE" %
%   B23:0/13  "PRIME MODE" %
%   T24:36  "FLIGHT DETECTED TIMER" %
%   B12:4/1  DO207  "O:2/7 MAIN CYL #7 DEPOSIT" %
%   T24:46  "SERVO GO SIGNAL HOLD TIMER" %
%   B23:0/0  ESTOP_OK  "E-STOP O.K." %
% Rung: 38 %
% MAIN CYL #8 %
SOR BST BST XIC B23:10/7 NXB XIC B23:0/13 BND XIC T24:37/DN NXB XIC B12:4/2 BND XIO T24:47/DN XIC B23:0/0 OTE B12:4/2 EOR
%   B23:10/7  "DEPOSIT POSITION #8 ACTIVE" %
%   B23:0/13  "PRIME MODE" %
%   T24:37  "READY FOR CUSTOMER PAN TIMER" %
%   B12:4/2  DO208  "O:2/8 MAIN CYL #8 DEPOSIT" %
%   T24:47  "JOG DELAY TIMER" %
%   B23:0/0  ESTOP_OK  "E-STOP O.K." %
% Rung: 39 %
% FILLER DEPOSIT IN PROGRESS %
SOR XIC B23:0/13 OTE B12:3/4 EOR
%   B23:0/13  "PRIME MODE" %
%   B12:3/4  DO02  "PROD VALVE IN DEPOSIT POSITION" %

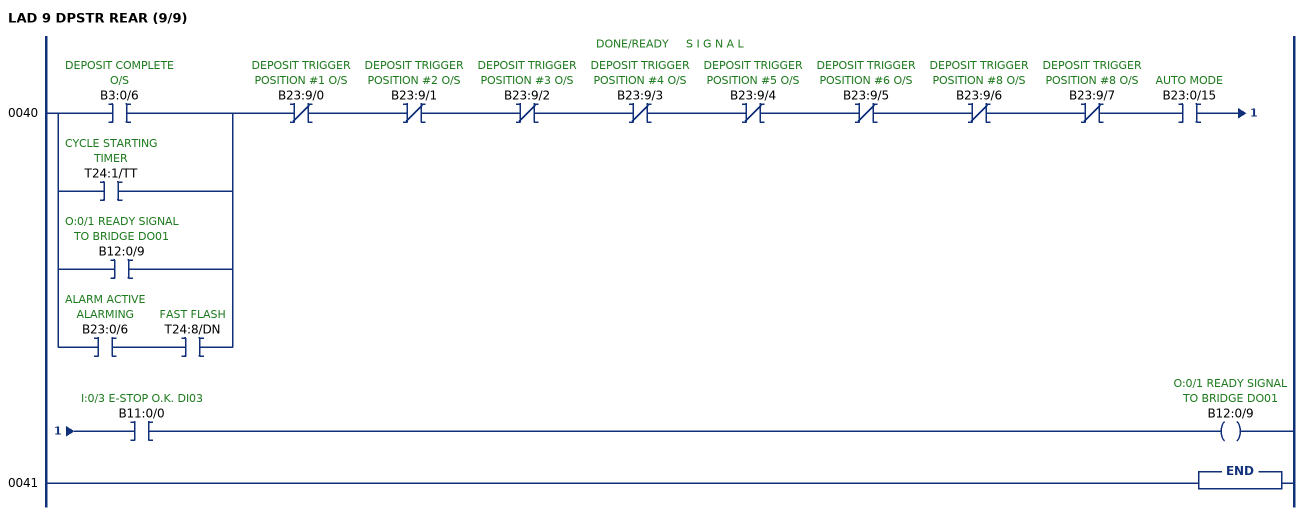
% Rung: 40 %
%         DONE/READY     S I G N A L %
SOR BST XIC B3:0/6 NXB XIC T24:1/TT NXB XIC B12:0/9 NXB XIC B23:0/6 XIC T24:8/DN BND XIO B23:9/0 XIO B23:9/1 XIO B23:9/2 XIO B23:9/3 XIO B23:9/4 XIO B23:9/5 XIO B23:9/6 XIO B23:9/7 XIC B23:0/15 XIC B11:0/0 OTE B12:0/9 EOR
%   B3:0/6  "DEPOSIT COMPLETE O/S" %
%   T24:1  "CYCLE STARTING TIMER" %
%   B12:0/9  DO01  "O:0/1 READY SIGNAL TO BRIDGE" %
%   B23:0/6  ALARMING  "ALARM ACTIVE" %
%   T24:8  "FAST FLASH" %
%   B23:9/0  "DEPOSIT TRIGGER POSITION #1 O/S" %
%   B23:9/1  "DEPOSIT TRIGGER POSITION #2 O/S" %
%   B23:9/2  "DEPOSIT TRIGGER POSITION #3 O/S" %
%   B23:9/3  "DEPOSIT TRIGGER POSITION #4 O/S" %
%   B23:9/4  "DEPOSIT TRIGGER POSITION #5 O/S" %
%   B23:9/5  "DEPOSIT TRIGGER POSITION #6 O/S" %
%   B23:9/6  "DEPOSIT TRIGGER POSITION #8 O/S" %
%   B23:9/7  "DEPOSIT TRIGGER POSITION #8 O/S" %
%   B23:0/15  "AUTO MODE" %
%   B11:0/0  DI03  "I:0/3 E-STOP O.K." %
% Rung: 41 %
SOR END EOR

LADDER 11 "MAP DI"
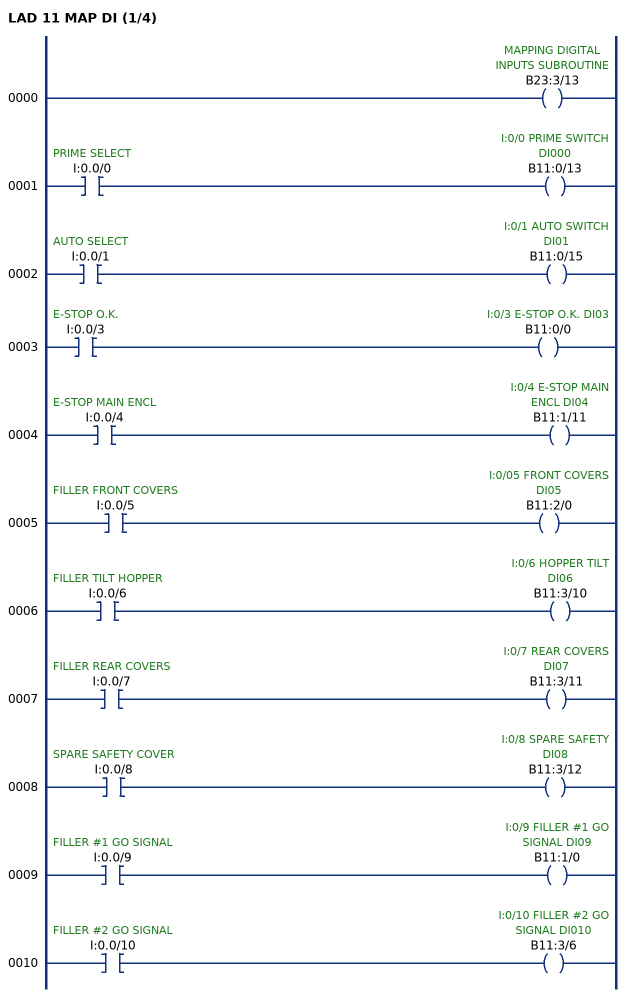
% Rung: 0 %
SOR OTE B23:3/13 EOR
%   B23:3/13  "MAPPING DIGITAL INPUTS SUBROUTINE" %
% Rung: 1 %
SOR XIC I:0.0/0 OTE B11:0/13 EOR
%   I:0.0/0  "PRIME SELECT" %
%   B11:0/13  DI000  "I:0/0 PRIME SWITCH" %
% Rung: 2 %
SOR XIC I:0.0/1 OTE B11:0/15 EOR
%   I:0.0/1  "AUTO SELECT" %
%   B11:0/15  DI01  "I:0/1 AUTO SWITCH" %
% Rung: 3 %
SOR XIC I:0.0/3 OTE B11:0/0 EOR
%   I:0.0/3  "E-STOP O.K." %
%   B11:0/0  DI03  "I:0/3 E-STOP O.K." %
% Rung: 4 %
SOR XIC I:0.0/4 OTE B11:1/11 EOR
%   I:0.0/4  "E-STOP MAIN ENCL" %
%   B11:1/11  DI04  "I:0/4 E-STOP MAIN ENCL" %
% Rung: 5 %
SOR XIC I:0.0/5 OTE B11:2/0 EOR
%   I:0.0/5  "FILLER FRONT COVERS" %
%   B11:2/0  DI05  "I:0/05 FRONT COVERS" %
% Rung: 6 %
SOR XIC I:0.0/6 OTE B11:3/10 EOR
%   I:0.0/6  "FILLER TILT HOPPER" %
%   B11:3/10  DI06  "I:0/6 HOPPER TILT" %
% Rung: 7 %
SOR XIC I:0.0/7 OTE B11:3/11 EOR
%   I:0.0/7  "FILLER REAR COVERS" %
%   B11:3/11  DI07  "I:0/7 REAR COVERS" %
% Rung: 8 %
SOR XIC I:0.0/8 OTE B11:3/12 EOR
%   I:0.0/8  "SPARE SAFETY COVER" %
%   B11:3/12  DI08  "I:0/8 SPARE SAFETY" %
% Rung: 9 %
SOR XIC I:0.0/9 OTE B11:1/0 EOR
%   I:0.0/9  "FILLER #1 GO SIGNAL" %
%   B11:1/0  DI09  "I:0/9 FILLER #1 GO SIGNAL" %
% Rung: 10 %
SOR XIC I:0.0/10 OTE B11:3/6 EOR
%   I:0.0/10  "FILLER #2 GO SIGNAL" %
%   B11:3/6  DI010  "I:0/10 FILLER #2 GO SIGNAL" %

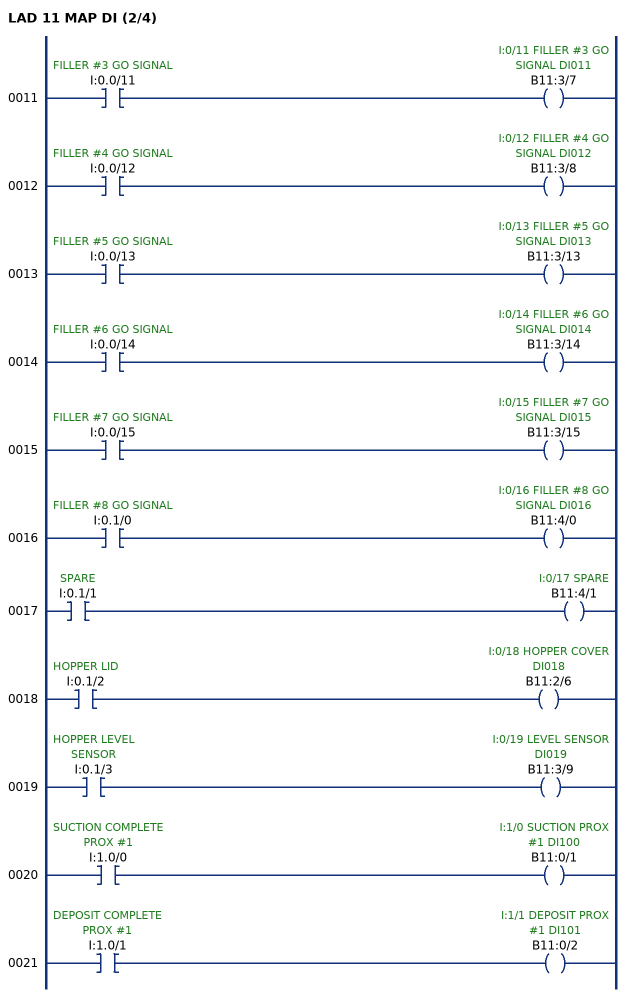
% Rung: 11 %
SOR XIC I:0.0/11 OTE B11:3/7 EOR
%   I:0.0/11  "FILLER #3 GO SIGNAL" %
%   B11:3/7  DI011  "I:0/11 FILLER #3 GO SIGNAL" %
% Rung: 12 %
SOR XIC I:0.0/12 OTE B11:3/8 EOR
%   I:0.0/12  "FILLER #4 GO SIGNAL" %
%   B11:3/8  DI012  "I:0/12 FILLER #4 GO SIGNAL" %
% Rung: 13 %
SOR XIC I:0.0/13 OTE B11:3/13 EOR
%   I:0.0/13  "FILLER #5 GO SIGNAL" %
%   B11:3/13  DI013  "I:0/13 FILLER #5 GO SIGNAL" %
% Rung: 14 %
SOR XIC I:0.0/14 OTE B11:3/14 EOR
%   I:0.0/14  "FILLER #6 GO SIGNAL" %
%   B11:3/14  DI014  "I:0/14 FILLER #6 GO SIGNAL" %
% Rung: 15 %
SOR XIC I:0.0/15 OTE B11:3/15 EOR
%   I:0.0/15  "FILLER #7 GO SIGNAL" %
%   B11:3/15  DI015  "I:0/15 FILLER #7 GO SIGNAL" %
% Rung: 16 %
SOR XIC I:0.1/0 OTE B11:4/0 EOR
%   I:0.1/0  "FILLER #8 GO SIGNAL" %
%   B11:4/0  DI016  "I:0/16 FILLER #8 GO SIGNAL" %
% Rung: 17 %
SOR XIC I:0.1/1 OTE B11:4/1 EOR
%   I:0.1/1  "SPARE" %
%   B11:4/1  "I:0/17 SPARE" %
% Rung: 18 %
SOR XIC I:0.1/2 OTE B11:2/6 EOR
%   I:0.1/2  "HOPPER LID" %
%   B11:2/6  DI018  "I:0/18 HOPPER COVER" %
% Rung: 19 %
SOR XIC I:0.1/3 OTE B11:3/9 EOR
%   I:0.1/3  "HOPPER LEVEL SENSOR" %
%   B11:3/9  DI019  "I:0/19 LEVEL SENSOR" %
% Rung: 20 %
SOR XIC I:1.0/0 OTE B11:0/1 EOR
%   I:1.0/0  "SUCTION COMPLETE PROX #1" %
%   B11:0/1  DI100  "I:1/0 SUCTION PROX #1" %
% Rung: 21 %
SOR XIC I:1.0/1 OTE B11:0/2 EOR
%   I:1.0/1  "DEPOSIT COMPLETE PROX #1" %
%   B11:0/2  DI101  "I:1/1 DEPOSIT PROX #1" %

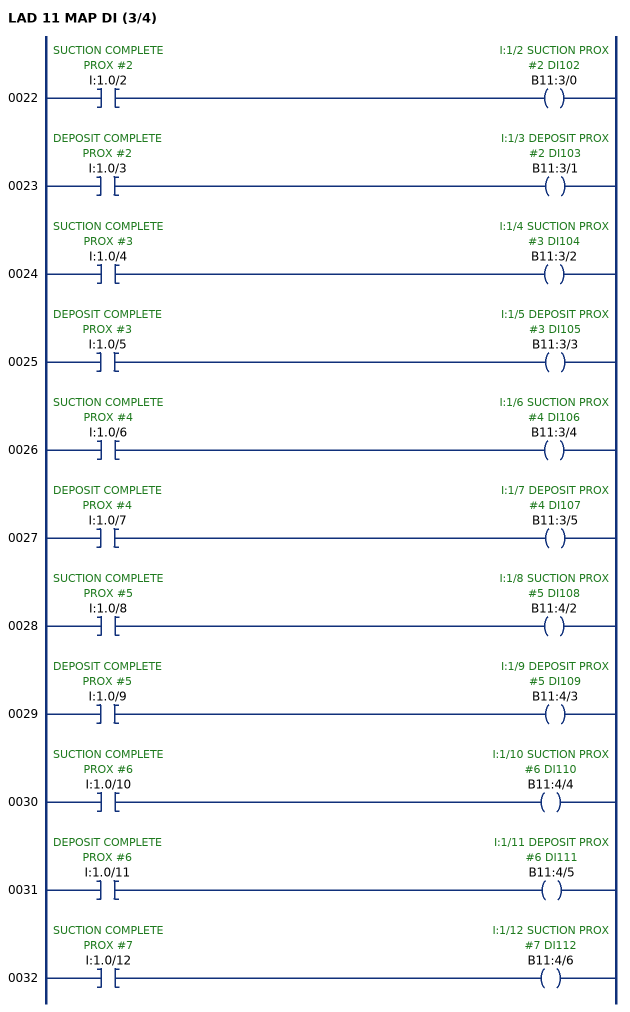
% Rung: 22 %
SOR XIC I:1.0/2 OTE B11:3/0 EOR
%   I:1.0/2  "SUCTION COMPLETE PROX #2" %
%   B11:3/0  DI102  "I:1/2 SUCTION PROX #2" %
% Rung: 23 %
SOR XIC I:1.0/3 OTE B11:3/1 EOR
%   I:1.0/3  "DEPOSIT COMPLETE PROX #2" %
%   B11:3/1  DI103  "I:1/3 DEPOSIT PROX #2" %
% Rung: 24 %
SOR XIC I:1.0/4 OTE B11:3/2 EOR
%   I:1.0/4  "SUCTION COMPLETE PROX #3" %
%   B11:3/2  DI104  "I:1/4 SUCTION PROX #3" %
% Rung: 25 %
SOR XIC I:1.0/5 OTE B11:3/3 EOR
%   I:1.0/5  "DEPOSIT COMPLETE PROX #3" %
%   B11:3/3  DI105  "I:1/5 DEPOSIT PROX #3" %
% Rung: 26 %
SOR XIC I:1.0/6 OTE B11:3/4 EOR
%   I:1.0/6  "SUCTION COMPLETE PROX #4" %
%   B11:3/4  DI106  "I:1/6 SUCTION PROX #4" %
% Rung: 27 %
SOR XIC I:1.0/7 OTE B11:3/5 EOR
%   I:1.0/7  "DEPOSIT COMPLETE PROX #4" %
%   B11:3/5  DI107  "I:1/7 DEPOSIT PROX #4" %
% Rung: 28 %
SOR XIC I:1.0/8 OTE B11:4/2 EOR
%   I:1.0/8  "SUCTION COMPLETE PROX #5" %
%   B11:4/2  DI108  "I:1/8 SUCTION PROX #5" %
% Rung: 29 %
SOR XIC I:1.0/9 OTE B11:4/3 EOR
%   I:1.0/9  "DEPOSIT COMPLETE PROX #5" %
%   B11:4/3  DI109  "I:1/9 DEPOSIT PROX #5" %
% Rung: 30 %
SOR XIC I:1.0/10 OTE B11:4/4 EOR
%   I:1.0/10  "SUCTION COMPLETE PROX #6" %
%   B11:4/4  DI110  "I:1/10 SUCTION PROX #6" %
% Rung: 31 %
SOR XIC I:1.0/11 OTE B11:4/5 EOR
%   I:1.0/11  "DEPOSIT COMPLETE PROX #6" %
%   B11:4/5  DI111  "I:1/11 DEPOSIT PROX #6" %
% Rung: 32 %
SOR XIC I:1.0/12 OTE B11:4/6 EOR
%   I:1.0/12  "SUCTION COMPLETE PROX #7" %
%   B11:4/6  DI112  "I:1/12 SUCTION PROX #7" %

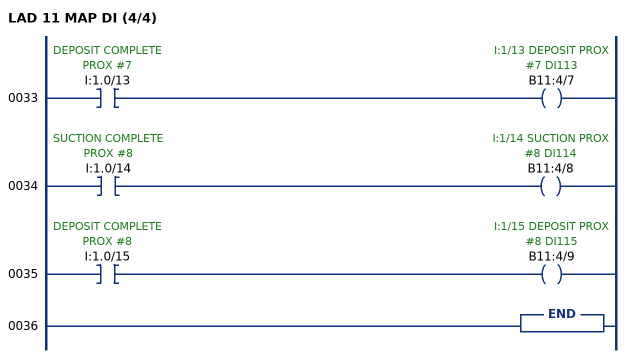
% Rung: 33 %
SOR XIC I:1.0/13 OTE B11:4/7 EOR
%   I:1.0/13  "DEPOSIT COMPLETE PROX #7" %
%   B11:4/7  DI113  "I:1/13 DEPOSIT PROX #7" %
% Rung: 34 %
SOR XIC I:1.0/14 OTE B11:4/8 EOR
%   I:1.0/14  "SUCTION COMPLETE PROX #8" %
%   B11:4/8  DI114  "I:1/14 SUCTION PROX #8" %
% Rung: 35 %
SOR XIC I:1.0/15 OTE B11:4/9 EOR
%   I:1.0/15  "DEPOSIT COMPLETE PROX #8" %
%   B11:4/9  DI115  "I:1/15 DEPOSIT PROX #8" %
% Rung: 36 %
SOR END EOR

LADDER 12 "MAP DO"
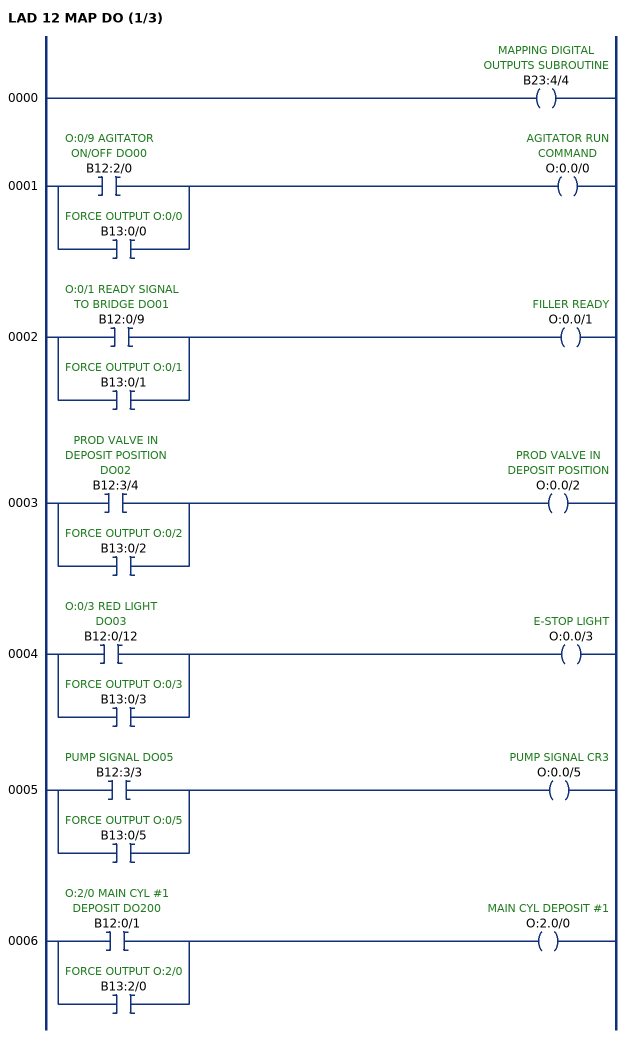
% Rung: 0 %
SOR OTE B23:4/4 EOR
%   B23:4/4  "MAPPING DIGITAL OUTPUTS SUBROUTINE" %
% Rung: 1 %
SOR BST XIC B12:2/0 NXB XIC B13:0/0 BND OTE O:0.0/0 EOR
%   B12:2/0  DO00  "O:0/9 AGITATOR ON/OFF" %
%   B13:0/0  "FORCE OUTPUT O:0/0" %
%   O:0.0/0  "AGITATOR RUN COMMAND" %
% Rung: 2 %
SOR BST XIC B12:0/9 NXB XIC B13:0/1 BND OTE O:0.0/1 EOR
%   B12:0/9  DO01  "O:0/1 READY SIGNAL TO BRIDGE" %
%   B13:0/1  "FORCE OUTPUT O:0/1" %
%   O:0.0/1  "FILLER READY" %
% Rung: 3 %
SOR BST XIC B12:3/4 NXB XIC B13:0/2 BND OTE O:0.0/2 EOR
%   B12:3/4  DO02  "PROD VALVE IN DEPOSIT POSITION" %
%   B13:0/2  "FORCE OUTPUT O:0/2" %
%   O:0.0/2  "PROD VALVE IN DEPOSIT POSITION" %
% Rung: 4 %
SOR BST XIC B12:0/12 NXB XIC B13:0/3 BND OTE O:0.0/3 EOR
%   B12:0/12  DO03  "O:0/3 RED LIGHT" %
%   B13:0/3  "FORCE OUTPUT O:0/3" %
%   O:0.0/3  "E-STOP LIGHT" %
% Rung: 5 %
SOR BST XIC B12:3/3 NXB XIC B13:0/5 BND OTE O:0.0/5 EOR
%   B12:3/3  DO05  "PUMP SIGNAL" %
%   B13:0/5  "FORCE OUTPUT O:0/5" %
%   O:0.0/5  "PUMP SIGNAL CR3" %
% Rung: 6 %
SOR BST XIC B12:0/1 NXB XIC B13:2/0 BND OTE O:2.0/0 EOR
%   B12:0/1  DO200  "O:2/0 MAIN CYL #1 DEPOSIT" %
%   B13:2/0  "FORCE OUTPUT O:2/0" %
%   O:2.0/0  "MAIN CYL DEPOSIT #1" %

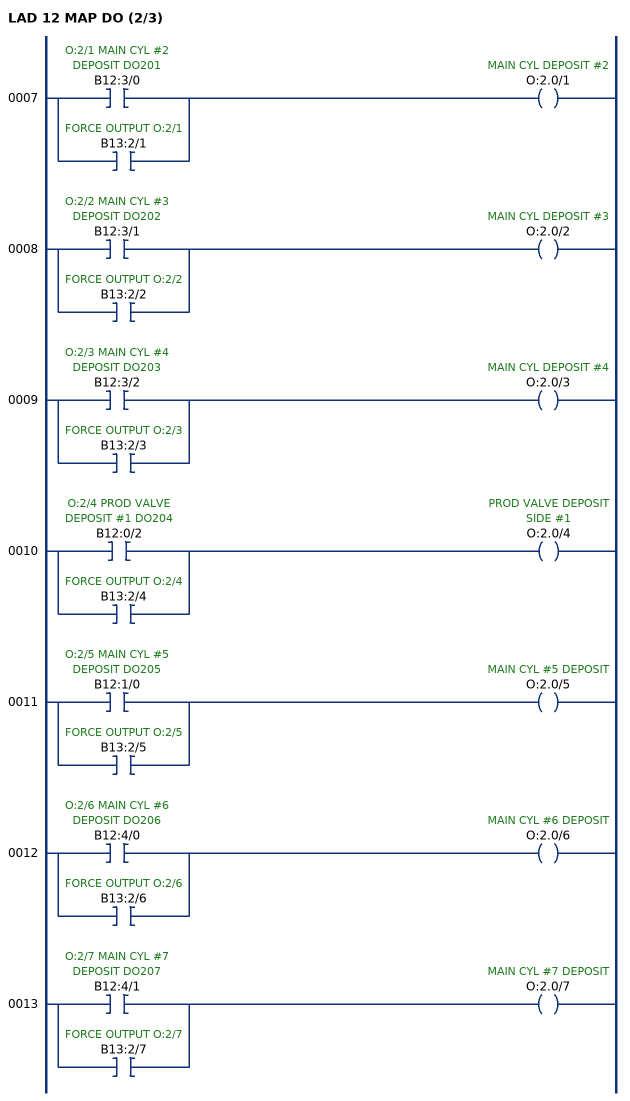
% Rung: 7 %
SOR BST XIC B12:3/0 NXB XIC B13:2/1 BND OTE O:2.0/1 EOR
%   B12:3/0  DO201  "O:2/1 MAIN CYL #2 DEPOSIT" %
%   B13:2/1  "FORCE OUTPUT O:2/1" %
%   O:2.0/1  "MAIN CYL DEPOSIT #2" %
% Rung: 8 %
SOR BST XIC B12:3/1 NXB XIC B13:2/2 BND OTE O:2.0/2 EOR
%   B12:3/1  DO202  "O:2/2 MAIN CYL #3 DEPOSIT" %
%   B13:2/2  "FORCE OUTPUT O:2/2" %
%   O:2.0/2  "MAIN CYL DEPOSIT #3" %
% Rung: 9 %
SOR BST XIC B12:3/2 NXB XIC B13:2/3 BND OTE O:2.0/3 EOR
%   B12:3/2  DO203  "O:2/3 MAIN CYL #4 DEPOSIT" %
%   B13:2/3  "FORCE OUTPUT O:2/3" %
%   O:2.0/3  "MAIN CYL DEPOSIT #4" %
% Rung: 10 %
SOR BST XIC B12:0/2 NXB XIC B13:2/4 BND OTE O:2.0/4 EOR
%   B12:0/2  DO204  "O:2/4 PROD VALVE DEPOSIT #1" %
%   B13:2/4  "FORCE OUTPUT O:2/4" %
%   O:2.0/4  "PROD VALVE DEPOSIT SIDE #1" %
% Rung: 11 %
SOR BST XIC B12:1/0 NXB XIC B13:2/5 BND OTE O:2.0/5 EOR
%   B12:1/0  DO205  "O:2/5 MAIN CYL #5 DEPOSIT" %
%   B13:2/5  "FORCE OUTPUT O:2/5" %
%   O:2.0/5  "MAIN CYL #5 DEPOSIT" %
% Rung: 12 %
SOR BST XIC B12:4/0 NXB XIC B13:2/6 BND OTE O:2.0/6 EOR
%   B12:4/0  DO206  "O:2/6 MAIN CYL #6 DEPOSIT" %
%   B13:2/6  "FORCE OUTPUT O:2/6" %
%   O:2.0/6  "MAIN CYL #6 DEPOSIT" %
% Rung: 13 %
SOR BST XIC B12:4/1 NXB XIC B13:2/7 BND OTE O:2.0/7 EOR
%   B12:4/1  DO207  "O:2/7 MAIN CYL #7 DEPOSIT" %
%   B13:2/7  "FORCE OUTPUT O:2/7" %
%   O:2.0/7  "MAIN CYL #7 DEPOSIT" %

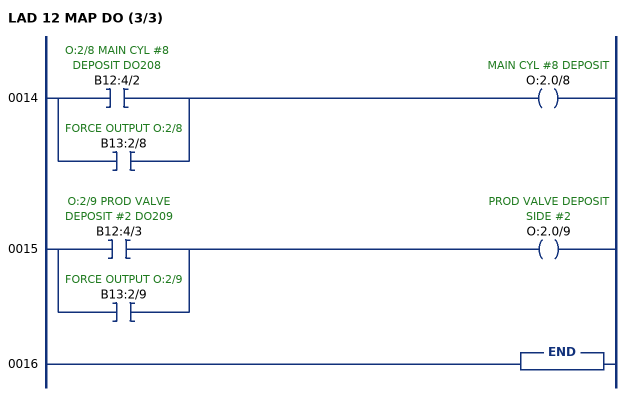
% Rung: 14 %
SOR BST XIC B12:4/2 NXB XIC B13:2/8 BND OTE O:2.0/8 EOR
%   B12:4/2  DO208  "O:2/8 MAIN CYL #8 DEPOSIT" %
%   B13:2/8  "FORCE OUTPUT O:2/8" %
%   O:2.0/8  "MAIN CYL #8 DEPOSIT" %
% Rung: 15 %
SOR BST XIC B12:4/3 NXB XIC B13:2/9 BND OTE O:2.0/9 EOR
%   B12:4/3  DO209  "O:2/9 PROD VALVE DEPOSIT #2" %
%   B13:2/9  "FORCE OUTPUT O:2/9" %
%   O:2.0/9  "PROD VALVE DEPOSIT SIDE #2" %
% Rung: 16 %
SOR END EOR

LADDER 14 "ALARMS"
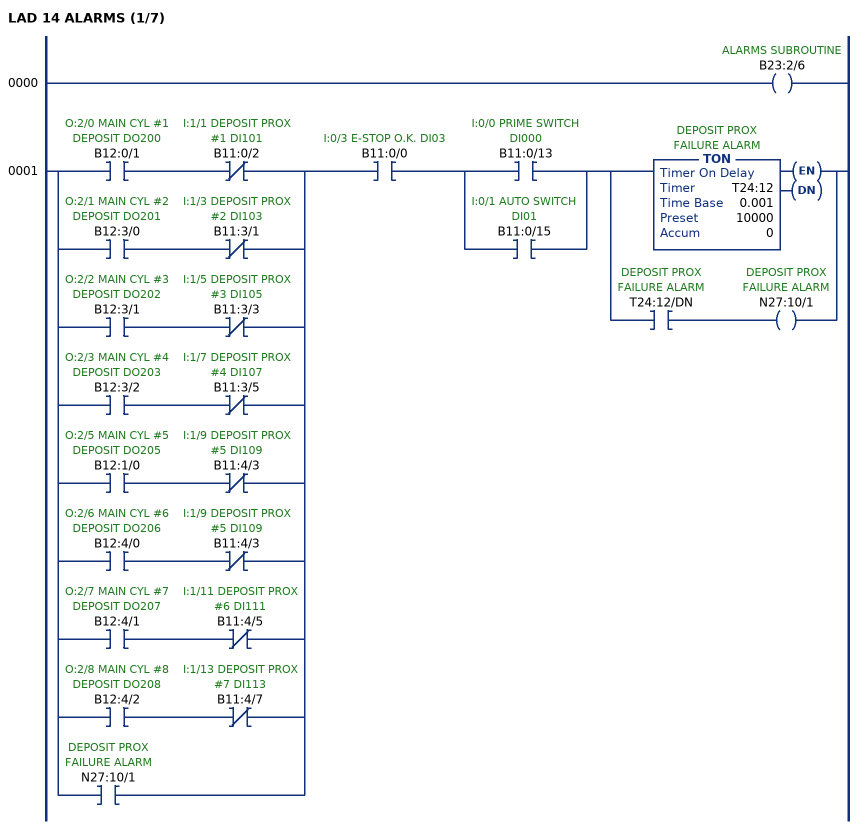
% Rung: 0 %
SOR OTE B23:2/6 EOR
%   B23:2/6  "ALARMS SUBROUTINE" %
% Rung: 1 %
SOR BST XIC B12:0/1 XIO B11:0/2 NXB XIC B12:3/0 XIO B11:3/1 NXB XIC B12:3/1 XIO B11:3/3 NXB XIC B12:3/2 XIO B11:3/5 NXB XIC B12:1/0 XIO B11:4/3 NXB XIC B12:4/0 XIO B11:4/3 NXB XIC B12:4/1 XIO B11:4/5 NXB XIC B12:4/2 XIO B11:4/7 NXB XIC N27:10/1 BND XIC B11:0/0 BST XIC B11:0/13 NXB XIC B11:0/15 BND BST TON T24:12 0.001 10000 0 NXB XIC T24:12/DN OTE N27:10/1 BND EOR
%   B12:0/1  DO200  "O:2/0 MAIN CYL #1 DEPOSIT" %
%   B11:0/2  DI101  "I:1/1 DEPOSIT PROX #1" %
%   B12:3/0  DO201  "O:2/1 MAIN CYL #2 DEPOSIT" %
%   B11:3/1  DI103  "I:1/3 DEPOSIT PROX #2" %
%   B12:3/1  DO202  "O:2/2 MAIN CYL #3 DEPOSIT" %
%   B11:3/3  DI105  "I:1/5 DEPOSIT PROX #3" %
%   B12:3/2  DO203  "O:2/3 MAIN CYL #4 DEPOSIT" %
%   B11:3/5  DI107  "I:1/7 DEPOSIT PROX #4" %
%   B12:1/0  DO205  "O:2/5 MAIN CYL #5 DEPOSIT" %
%   B11:4/3  DI109  "I:1/9 DEPOSIT PROX #5" %
%   B12:4/0  DO206  "O:2/6 MAIN CYL #6 DEPOSIT" %
%   B12:4/1  DO207  "O:2/7 MAIN CYL #7 DEPOSIT" %
%   B11:4/5  DI111  "I:1/11 DEPOSIT PROX #6" %
%   B12:4/2  DO208  "O:2/8 MAIN CYL #8 DEPOSIT" %
%   B11:4/7  DI113  "I:1/13 DEPOSIT PROX #7" %
%   N27:10/1  "DEPOSIT PROX FAILURE ALARM" %
%   B11:0/0  DI03  "I:0/3 E-STOP O.K." %
%   B11:0/13  DI000  "I:0/0 PRIME SWITCH" %
%   B11:0/15  DI01  "I:0/1 AUTO SWITCH" %
%   T24:12  "DEPOSIT PROX FAILURE ALARM" %

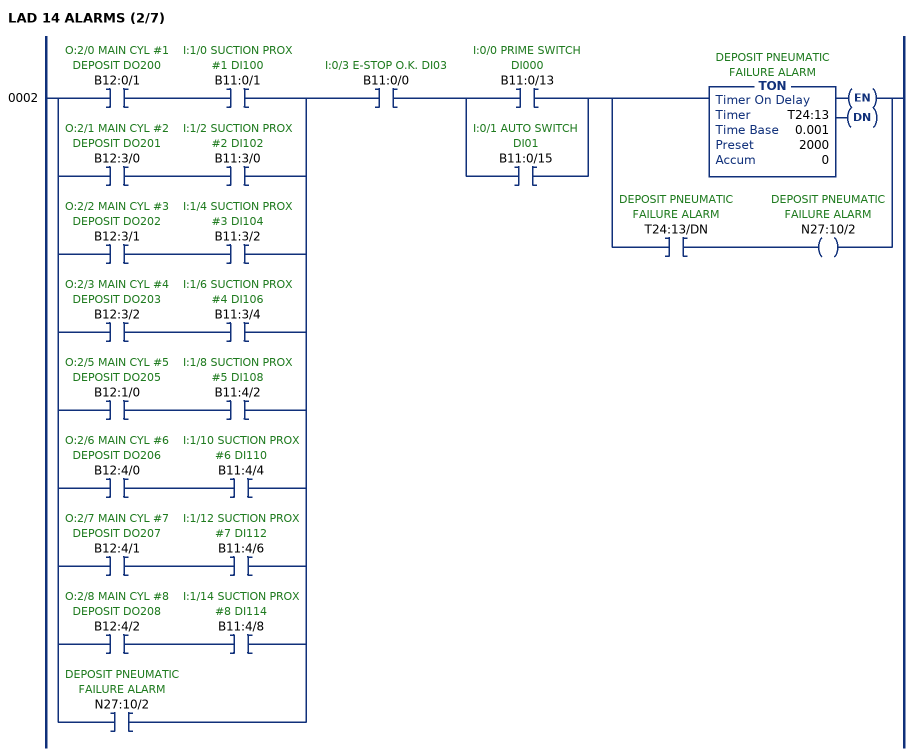
% Rung: 2 %
SOR BST XIC B12:0/1 XIC B11:0/1 NXB XIC B12:3/0 XIC B11:3/0 NXB XIC B12:3/1 XIC B11:3/2 NXB XIC B12:3/2 XIC B11:3/4 NXB XIC B12:1/0 XIC B11:4/2 NXB XIC B12:4/0 XIC B11:4/4 NXB XIC B12:4/1 XIC B11:4/6 NXB XIC B12:4/2 XIC B11:4/8 NXB XIC N27:10/2 BND XIC B11:0/0 BST XIC B11:0/13 NXB XIC B11:0/15 BND BST TON T24:13 0.001 2000 0 NXB XIC T24:13/DN OTE N27:10/2 BND EOR
%   B12:0/1  DO200  "O:2/0 MAIN CYL #1 DEPOSIT" %
%   B11:0/1  DI100  "I:1/0 SUCTION PROX #1" %
%   B12:3/0  DO201  "O:2/1 MAIN CYL #2 DEPOSIT" %
%   B11:3/0  DI102  "I:1/2 SUCTION PROX #2" %
%   B12:3/1  DO202  "O:2/2 MAIN CYL #3 DEPOSIT" %
%   B11:3/2  DI104  "I:1/4 SUCTION PROX #3" %
%   B12:3/2  DO203  "O:2/3 MAIN CYL #4 DEPOSIT" %
%   B11:3/4  DI106  "I:1/6 SUCTION PROX #4" %
%   B12:1/0  DO205  "O:2/5 MAIN CYL #5 DEPOSIT" %
%   B11:4/2  DI108  "I:1/8 SUCTION PROX #5" %
%   B12:4/0  DO206  "O:2/6 MAIN CYL #6 DEPOSIT" %
%   B11:4/4  DI110  "I:1/10 SUCTION PROX #6" %
%   B12:4/1  DO207  "O:2/7 MAIN CYL #7 DEPOSIT" %
%   B11:4/6  DI112  "I:1/12 SUCTION PROX #7" %
%   B12:4/2  DO208  "O:2/8 MAIN CYL #8 DEPOSIT" %
%   B11:4/8  DI114  "I:1/14 SUCTION PROX #8" %
%   N27:10/2  "DEPOSIT PNEUMATIC FAILURE ALARM" %
%   B11:0/0  DI03  "I:0/3 E-STOP O.K." %
%   B11:0/13  DI000  "I:0/0 PRIME SWITCH" %
%   B11:0/15  DI01  "I:0/1 AUTO SWITCH" %
%   T24:13  "DEPOSIT PNEUMATIC FAILURE ALARM" %

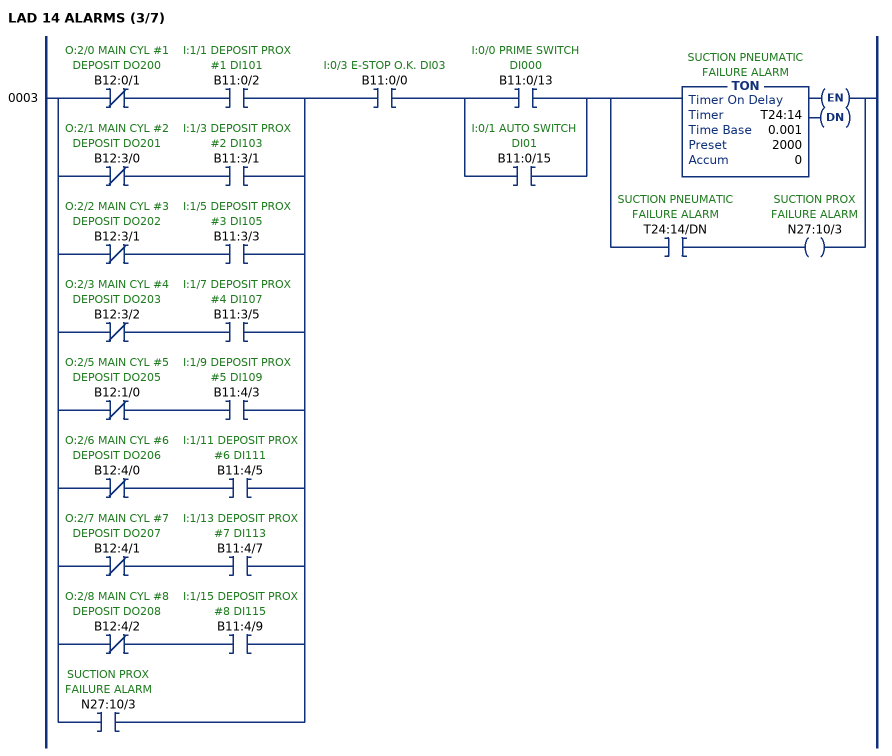
% Rung: 3 %
SOR BST XIO B12:0/1 XIC B11:0/2 NXB XIO B12:3/0 XIC B11:3/1 NXB XIO B12:3/1 XIC B11:3/3 NXB XIO B12:3/2 XIC B11:3/5 NXB XIO B12:1/0 XIC B11:4/3 NXB XIO B12:4/0 XIC B11:4/5 NXB XIO B12:4/1 XIC B11:4/7 NXB XIO B12:4/2 XIC B11:4/9 NXB XIC N27:10/3 BND XIC B11:0/0 BST XIC B11:0/13 NXB XIC B11:0/15 BND BST TON T24:14 0.001 2000 0 NXB XIC T24:14/DN OTE N27:10/3 BND EOR
%   B12:0/1  DO200  "O:2/0 MAIN CYL #1 DEPOSIT" %
%   B11:0/2  DI101  "I:1/1 DEPOSIT PROX #1" %
%   B12:3/0  DO201  "O:2/1 MAIN CYL #2 DEPOSIT" %
%   B11:3/1  DI103  "I:1/3 DEPOSIT PROX #2" %
%   B12:3/1  DO202  "O:2/2 MAIN CYL #3 DEPOSIT" %
%   B11:3/3  DI105  "I:1/5 DEPOSIT PROX #3" %
%   B12:3/2  DO203  "O:2/3 MAIN CYL #4 DEPOSIT" %
%   B11:3/5  DI107  "I:1/7 DEPOSIT PROX #4" %
%   B12:1/0  DO205  "O:2/5 MAIN CYL #5 DEPOSIT" %
%   B11:4/3  DI109  "I:1/9 DEPOSIT PROX #5" %
%   B12:4/0  DO206  "O:2/6 MAIN CYL #6 DEPOSIT" %
%   B11:4/5  DI111  "I:1/11 DEPOSIT PROX #6" %
%   B12:4/1  DO207  "O:2/7 MAIN CYL #7 DEPOSIT" %
%   B11:4/7  DI113  "I:1/13 DEPOSIT PROX #7" %
%   B12:4/2  DO208  "O:2/8 MAIN CYL #8 DEPOSIT" %
%   B11:4/9  DI115  "I:1/15 DEPOSIT PROX #8" %
%   N27:10/3  "SUCTION PROX FAILURE ALARM" %
%   B11:0/0  DI03  "I:0/3 E-STOP O.K." %
%   B11:0/13  DI000  "I:0/0 PRIME SWITCH" %
%   B11:0/15  DI01  "I:0/1 AUTO SWITCH" %
%   T24:14  "SUCTION PNEUMATIC FAILURE ALARM" %

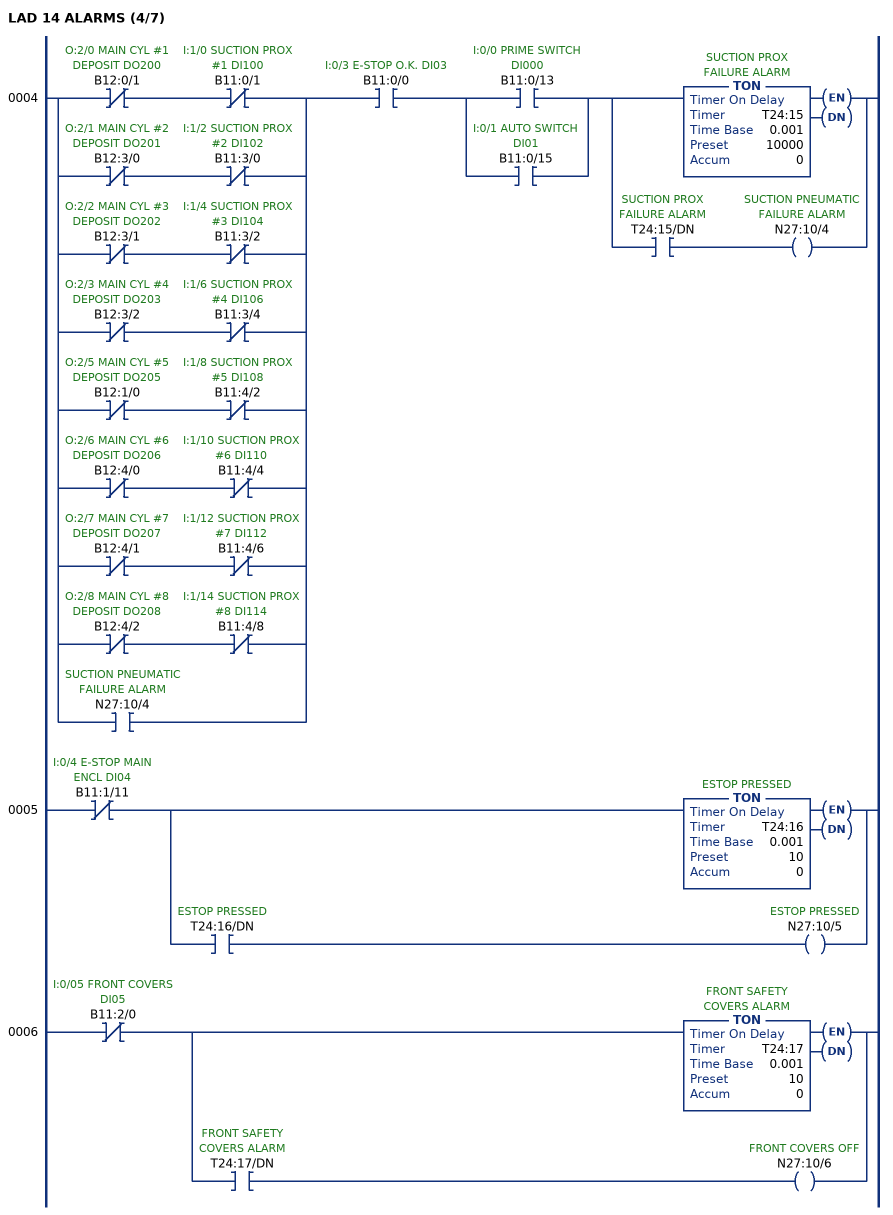
% Rung: 4 %
SOR BST XIO B12:0/1 XIO B11:0/1 NXB XIO B12:3/0 XIO B11:3/0 NXB XIO B12:3/1 XIO B11:3/2 NXB XIO B12:3/2 XIO B11:3/4 NXB XIO B12:1/0 XIO B11:4/2 NXB XIO B12:4/0 XIO B11:4/4 NXB XIO B12:4/1 XIO B11:4/6 NXB XIO B12:4/2 XIO B11:4/8 NXB XIC N27:10/4 BND XIC B11:0/0 BST XIC B11:0/13 NXB XIC B11:0/15 BND BST TON T24:15 0.001 10000 0 NXB XIC T24:15/DN OTE N27:10/4 BND EOR
%   B12:0/1  DO200  "O:2/0 MAIN CYL #1 DEPOSIT" %
%   B11:0/1  DI100  "I:1/0 SUCTION PROX #1" %
%   B12:3/0  DO201  "O:2/1 MAIN CYL #2 DEPOSIT" %
%   B11:3/0  DI102  "I:1/2 SUCTION PROX #2" %
%   B12:3/1  DO202  "O:2/2 MAIN CYL #3 DEPOSIT" %
%   B11:3/2  DI104  "I:1/4 SUCTION PROX #3" %
%   B12:3/2  DO203  "O:2/3 MAIN CYL #4 DEPOSIT" %
%   B11:3/4  DI106  "I:1/6 SUCTION PROX #4" %
%   B12:1/0  DO205  "O:2/5 MAIN CYL #5 DEPOSIT" %
%   B11:4/2  DI108  "I:1/8 SUCTION PROX #5" %
%   B12:4/0  DO206  "O:2/6 MAIN CYL #6 DEPOSIT" %
%   B11:4/4  DI110  "I:1/10 SUCTION PROX #6" %
%   B12:4/1  DO207  "O:2/7 MAIN CYL #7 DEPOSIT" %
%   B11:4/6  DI112  "I:1/12 SUCTION PROX #7" %
%   B12:4/2  DO208  "O:2/8 MAIN CYL #8 DEPOSIT" %
%   B11:4/8  DI114  "I:1/14 SUCTION PROX #8" %
%   N27:10/4  "SUCTION PNEUMATIC FAILURE ALARM" %
%   B11:0/0  DI03  "I:0/3 E-STOP O.K." %
%   B11:0/13  DI000  "I:0/0 PRIME SWITCH" %
%   B11:0/15  DI01  "I:0/1 AUTO SWITCH" %
%   T24:15  "SUCTION PROX FAILURE ALARM" %
% Rung: 5 %
SOR XIO B11:1/11 BST TON T24:16 0.001 10 0 NXB XIC T24:16/DN OTE N27:10/5 BND EOR
%   B11:1/11  DI04  "I:0/4 E-STOP MAIN ENCL" %
%   T24:16  "ESTOP PRESSED" %
%   N27:10/5  "ESTOP PRESSED" %
% Rung: 6 %
SOR XIO B11:2/0 BST TON T24:17 0.001 10 0 NXB XIC T24:17/DN OTE N27:10/6 BND EOR
%   B11:2/0  DI05  "I:0/05 FRONT COVERS" %
%   T24:17  "FRONT SAFETY COVERS ALARM" %
%   N27:10/6  "FRONT COVERS OFF" %

